      A     M      3.3;
      =     L     10.0;
      BLD   103;
      CALL FB    13 , DB    81 (
           EN_R                     := L     10.0,
           ID                       := W#16#1,
           R_ID                     := DW#16#1,
           NDR                      := DB2.DBX  100.0,
           ERROR                    := DB2.DBX  100.1,
           STATUS                   := DB2.DBW  102,
           RD_1                     := P#DB1.DBX0.0 BYTE 500,
           LEN                      := #RECV1_LEN);
      NOP   0;
NETWORK
TITLE =

      CALL SFC   20 (
           SRCBLK                   := P#M 5000.0 WORD 40,
           RET_VAL                  := #SFC20_RET_VAL,
           DSTBLK                   := P#DB21.DBX 0.0 WORD 40);
      NOP   0;
NETWORK
TITLE =

      L     80;
      T     #SEND1_LEN;
      NOP   0;
NETWORK
TITLE =LOCAL(CPU2) --> MAIN(CPU1) 공정상태

      A     M      0.2;
      =     L     10.0;
      BLD   103;
      AN    M      3.3;
      =     L     10.1;
      BLD   103;
      CALL FB    12 , DB    71 (
           REQ                      := L     10.0,
           R                        := L     10.1,
           ID                       := W#16#2,
           R_ID                     := DW#16#2,
           DONE                     := DB2.DBX    0.0,
           ERROR                    := DB2.DBX    0.1,
           STATUS                   := DB2.DBW    2,
           SD_1                     := P#DB21.DBX0.0 BYTE 80,
           LEN                      := #SEND1_LEN);
      NOP   0;
NETWORK
TITLE =

      L     80;
      T     #RECV2_LEN;
      NOP   0;
NETWORK
TITLE =MAIN(CPU1) --> LOCAL(CPU2) 셔틀상태
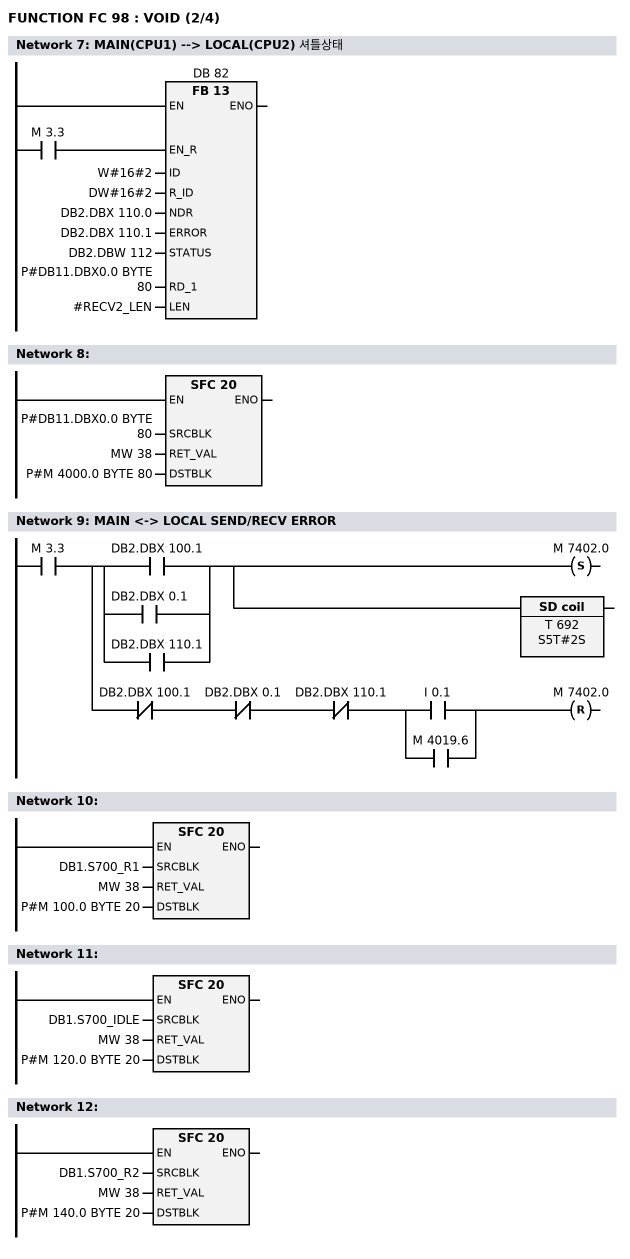

      A     M      3.3;
      =     L     10.0;
      BLD   103;
      CALL FB    13 , DB    82 (
           EN_R                     := L     10.0,
           ID                       := W#16#2,
           R_ID                     := DW#16#2,
           NDR                      := DB2.DBX  110.0,
           ERROR                    := DB2.DBX  110.1,
           STATUS                   := DB2.DBW  112,
           RD_1                     := P#DB11.DBX0.0 BYTE 80,
           LEN                      := #RECV2_LEN);
      NOP   0;
NETWORK
TITLE =

      CALL SFC   20 (
           SRCBLK                   := P#DB11.DBX0.0 BYTE 80,
           RET_VAL                  := MW    38,
           DSTBLK                   := P#M 4000.0 BYTE 80);
      NOP   0;
NETWORK
TITLE =MAIN <-> LOCAL SEND/RECV ERROR

      A     M      3.3;
      =     L     10.0;
      A     L     10.0;
      A(    ;
      O     DB2.DBX  100.1;
      O     DB2.DBX    0.1;
      O     DB2.DBX  110.1;
      )     ;
      S     M   7402.0;
      L     S5T#2S;
      SD    T    692;
      A     L     10.0;
      AN    DB2.DBX  100.1;
      AN    DB2.DBX    0.1;
      AN    DB2.DBX  110.1;
      A(    ;
      O     I      0.1;
      O     M   4019.6;
      )     ;
      R     M   7402.0;
NETWORK
TITLE =

      CALL SFC   20 (
           SRCBLK                   := DB1.S700_R1,
           RET_VAL                  := MW    38,
           DSTBLK                   := P#M 100.0 BYTE 20);
      NOP   0;
NETWORK
TITLE =

      CALL SFC   20 (
           SRCBLK                   := DB1.S700_IDLE,
           RET_VAL                  := MW    38,
           DSTBLK                   := P#M 120.0 BYTE 20);
      NOP   0;
NETWORK
TITLE =

      CALL SFC   20 (
           SRCBLK                   := DB1.S700_R2,
           RET_VAL                  := MW    38,
           DSTBLK                   := P#M 140.0 BYTE 20);
      NOP   0;
NETWORK
TITLE =
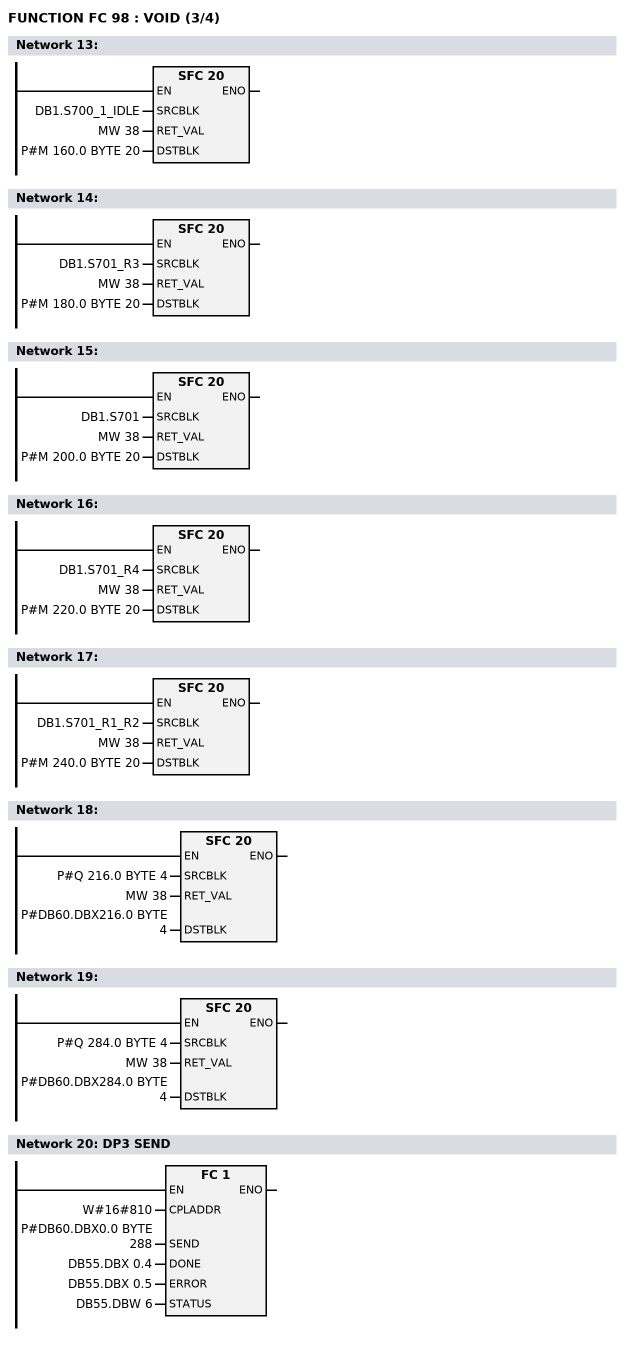

      CALL SFC   20 (
           SRCBLK                   := DB1.S700_1_IDLE,
           RET_VAL                  := MW    38,
           DSTBLK                   := P#M 160.0 BYTE 20);
      NOP   0;
NETWORK
TITLE =

      CALL SFC   20 (
           SRCBLK                   := DB1.S701_R3,
           RET_VAL                  := MW    38,
           DSTBLK                   := P#M 180.0 BYTE 20);
      NOP   0;
NETWORK
TITLE =

      CALL SFC   20 (
           SRCBLK                   := DB1.S701,
           RET_VAL                  := MW    38,
           DSTBLK                   := P#M 200.0 BYTE 20);
      NOP   0;
NETWORK
TITLE =

      CALL SFC   20 (
           SRCBLK                   := DB1.S701_R4,
           RET_VAL                  := MW    38,
           DSTBLK                   := P#M 220.0 BYTE 20);
      NOP   0;
NETWORK
TITLE =

      CALL SFC   20 (
           SRCBLK                   := DB1.S701_R1_R2,
           RET_VAL                  := MW    38,
           DSTBLK                   := P#M 240.0 BYTE 20);
      NOP   0;
NETWORK
TITLE =

      CALL SFC   20 (
           SRCBLK                   := P#Q 216.0 BYTE 4,
           RET_VAL                  := MW    38,
           DSTBLK                   := P#DB60.DBX216.0 BYTE 4);
      NOP   0;
NETWORK
TITLE =

      CALL SFC   20 (
           SRCBLK                   := P#Q 284.0 BYTE 4,
           RET_VAL                  := MW    38,
           DSTBLK                   := P#DB60.DBX284.0 BYTE 4);
      NOP   0;
NETWORK
TITLE =DP3 SEND

      CALL FC     1 (
           CPLADDR                  := W#16#810,
           SEND                     := P#DB60.DBX0.0 BYTE 288,
           DONE                     := DB55.DBX    0.4,
           ERROR                    := DB55.DBX    0.5,
           STATUS                   := DB55.DBW    6);
      NOP   0;
NETWORK
TITLE =DP3 RECV
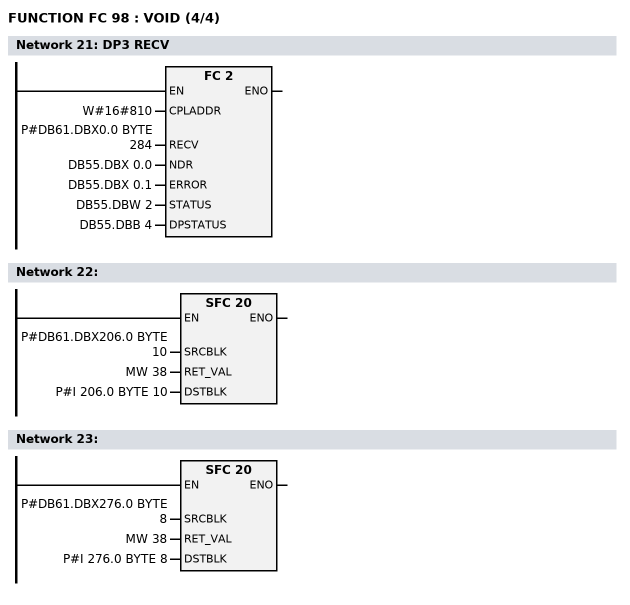

      CALL FC     2 (
           CPLADDR                  := W#16#810,
           RECV                     := P#DB61.DBX0.0 BYTE 284,
           NDR                      := DB55.DBX    0.0,
           ERROR                    := DB55.DBX    0.1,
           STATUS                   := DB55.DBW    2,
           DPSTATUS                 := DB55.DBB    4);
      NOP   0;
NETWORK
TITLE =

      CALL SFC   20 (
           SRCBLK                   := P#DB61.DBX206.0 BYTE 10,
           RET_VAL                  := MW    38,
           DSTBLK                   := P#I 206.0 BYTE 10);
      NOP   0;
NETWORK
TITLE =

      CALL SFC   20 (
           SRCBLK                   := P#DB61.DBX276.0 BYTE 8,
           RET_VAL                  := MW    38,
           DSTBLK                   := P#I 276.0 BYTE 8);
      NOP   0;
END_FUNCTION

FUNCTION FC 100 : VOID
TITLE =
VERSION : 0.1

BEGIN
NETWORK
TITLE =
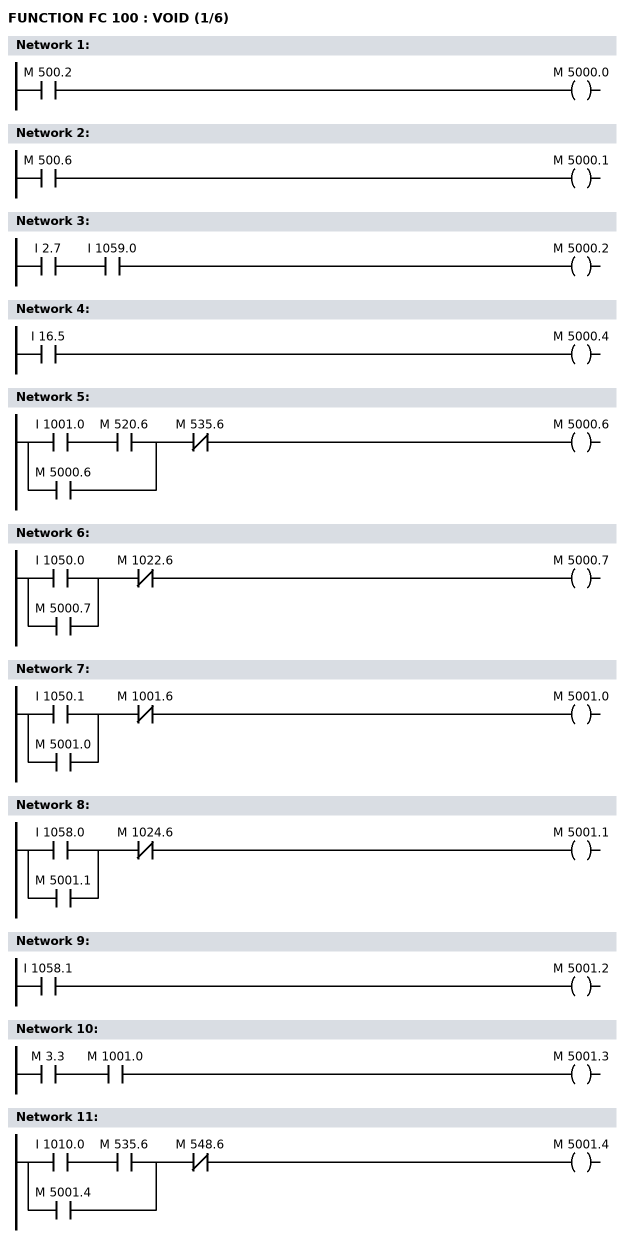

      A     M    500.2;
      =     M   5000.0;
NETWORK
TITLE =

      A     M    500.6;
      =     M   5000.1;
NETWORK
TITLE =

      A     I      2.7;
      A     I   1059.0;
      =     M   5000.2;
NETWORK
TITLE =

      A     I     16.5;
      =     M   5000.4;
NETWORK
TITLE =

      A(    ;
      A     I   1001.0;
      A     M    520.6;
      O     M   5000.6;
      )     ;
      AN    M    535.6;
      =     M   5000.6;
NETWORK
TITLE =

      A(    ;
      O     I   1050.0;
      O     M   5000.7;
      )     ;
      AN    M   1022.6;
      =     M   5000.7;
NETWORK
TITLE =

      A(    ;
      O     I   1050.1;
      O     M   5001.0;
      )     ;
      AN    M   1001.6;
      =     M   5001.0;
NETWORK
TITLE =

      A(    ;
      O     I   1058.0;
      O     M   5001.1;
      )     ;
      AN    M   1024.6;
      =     M   5001.1;
NETWORK
TITLE =

      A     I   1058.1;
      =     M   5001.2;
NETWORK
TITLE =

      A     M      3.3;
      A     M   1001.0;
      =     M   5001.3;
NETWORK
TITLE =

      A(    ;
      A     I   1010.0;
      A     M    535.6;
      O     M   5001.4;
      )     ;
      AN    M    548.6;
      =     M   5001.4;
NETWORK
TITLE =
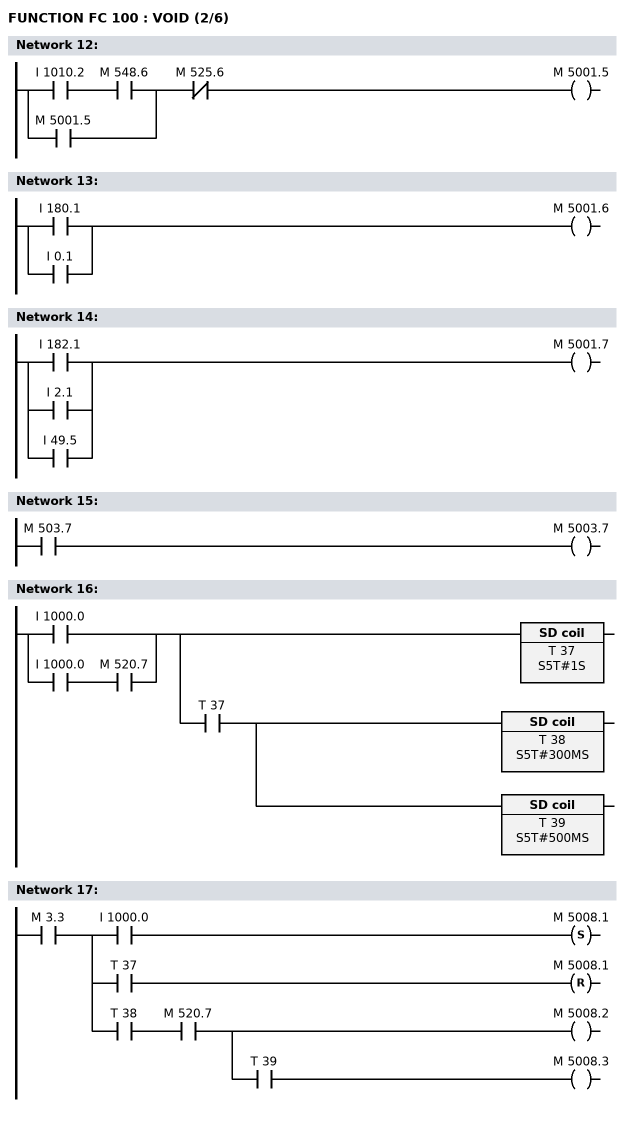

      A(    ;
      A     I   1010.2;
      A     M    548.6;
      O     M   5001.5;
      )     ;
      AN    M    525.6;
      =     M   5001.5;
NETWORK
TITLE =

      O     I    180.1;
      O     I      0.1;
      =     M   5001.6;
NETWORK
TITLE =

      O     I    182.1;
      O     I      2.1;
      O     I     49.5;
      =     M   5001.7;
NETWORK
TITLE =

      A     M    503.7;
      =     M   5003.7;
NETWORK
TITLE =

      O     I   1000.0;
      O     ;
      A     I   1000.0;
      A     M    520.7;
      =     L      0.0;
      A     L      0.0;
      BLD   102;
      L     S5T#1S;
      SD    T     37;
      A     L      0.0;
      A     T     37;
      L     S5T#300MS;
      SD    T     38;
      L     S5T#500MS;
      SD    T     39;
NETWORK
TITLE =

      A     M      3.3;
      =     L      0.0;
      A     L      0.0;
      A     I   1000.0;
      S     M   5008.1;
      A     L      0.0;
      A     T     37;
      R     M   5008.1;
      A     L      0.0;
      A     T     38;
      A     M    520.7;
      =     L      0.1;
      A     L      0.1;
      BLD   102;
      =     M   5008.2;
      A     L      0.1;
      A     T     39;
      =     M   5008.3;
NETWORK
TITLE =
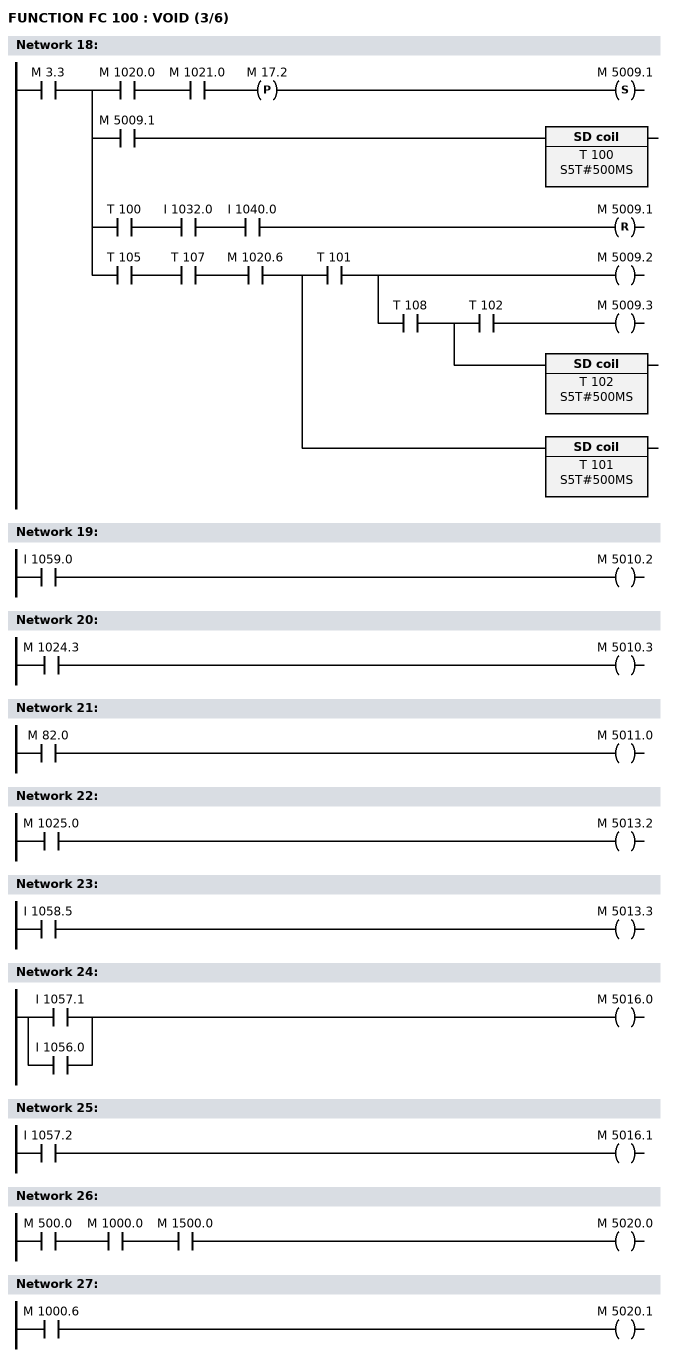

      A     M      3.3;
      =     L      0.0;
      A     L      0.0;
      A     M   1020.0;
      A     M   1021.0;
      FP    M     17.2;
      S     M   5009.1;
      A     L      0.0;
      A     M   5009.1;
      L     S5T#500MS;
      SD    T    100;
      A     L      0.0;
      A     T    100;
      A     I   1032.0;
      A     I   1040.0;
      R     M   5009.1;
      A     L      0.0;
      A     T    105;
      A     T    107;
      A     M   1020.6;
      =     L      0.1;
      A     L      0.1;
      A     T    101;
      =     L      0.2;
      A     L      0.2;
      BLD   102;
      =     M   5009.2;
      A     L      0.2;
      A     T    108;
      =     L      0.3;
      A     L      0.3;
      A     T    102;
      =     M   5009.3;
      A     L      0.3;
      BLD   102;
      L     S5T#500MS;
      SD    T    102;
      A     L      0.1;
      BLD   102;
      L     S5T#500MS;
      SD    T    101;
NETWORK
TITLE =

      A     I   1059.0;
      =     M   5010.2;
NETWORK
TITLE =

      A     M   1024.3;
      =     M   5010.3;
NETWORK
TITLE =

      A     M     82.0;
      =     M   5011.0;
NETWORK
TITLE =

      A     M   1025.0;
      =     M   5013.2;
NETWORK
TITLE =

      A     I   1058.5;
      =     M   5013.3;
NETWORK
TITLE =

      O     I   1057.1;
      O     I   1056.0;
      =     M   5016.0;
NETWORK
TITLE =

      A     I   1057.2;
      =     M   5016.1;
NETWORK
TITLE =

      A     M    500.0;
      A     M   1000.0;
      A     M   1500.0;
      =     M   5020.0;
NETWORK
TITLE =

      A     M   1000.6;
      =     M   5020.1;
NETWORK
TITLE =
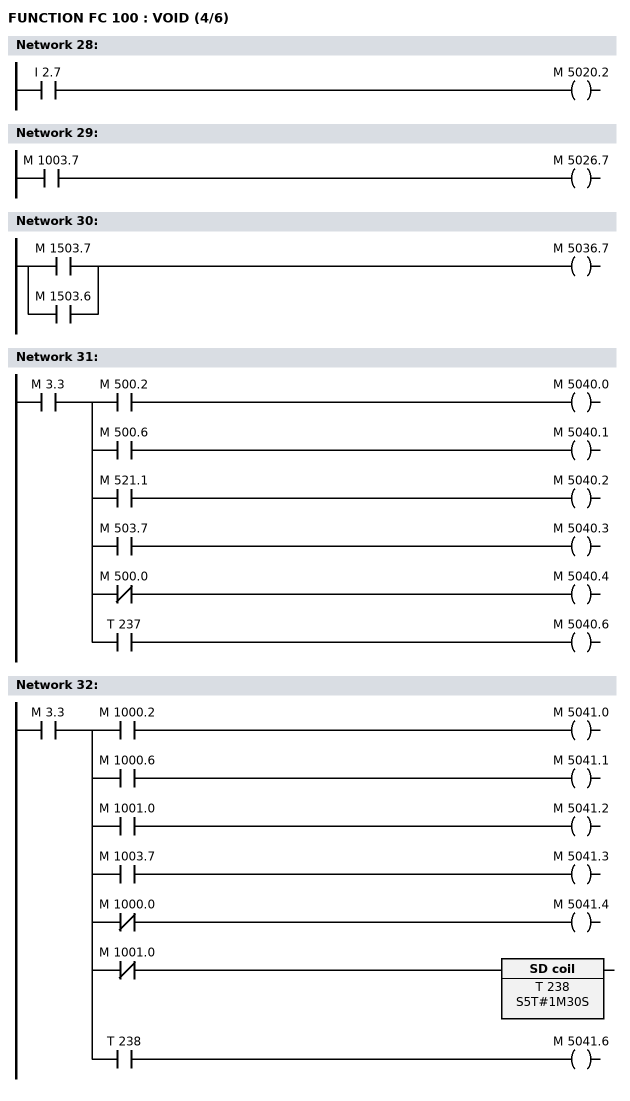

      A     I      2.7;
      =     M   5020.2;
NETWORK
TITLE =

      A     M   1003.7;
      =     M   5026.7;
NETWORK
TITLE =

      O     M   1503.7;
      O     M   1503.6;
      =     M   5036.7;
NETWORK
TITLE =

      A     M      3.3;
      =     L      0.0;
      A     L      0.0;
      A     M    500.2;
      =     M   5040.0;
      A     L      0.0;
      A     M    500.6;
      =     M   5040.1;
      A     L      0.0;
      A     M    521.1;
      =     M   5040.2;
      A     L      0.0;
      A     M    503.7;
      =     M   5040.3;
      A     L      0.0;
      AN    M    500.0;
      =     M   5040.4;
      A     L      0.0;
      A     T    237;
      =     M   5040.6;
NETWORK
TITLE =

      A     M      3.3;
      =     L      0.0;
      A     L      0.0;
      A     M   1000.2;
      =     M   5041.0;
      A     L      0.0;
      A     M   1000.6;
      =     M   5041.1;
      A     L      0.0;
      A     M   1001.0;
      =     M   5041.2;
      A     L      0.0;
      A     M   1003.7;
      =     M   5041.3;
      A     L      0.0;
      AN    M   1000.0;
      =     M   5041.4;
      A     L      0.0;
      AN    M   1001.0;
      L     S5T#1M30S;
      SD    T    238;
      A     L      0.0;
      A     T    238;
      =     M   5041.6;
NETWORK
TITLE =
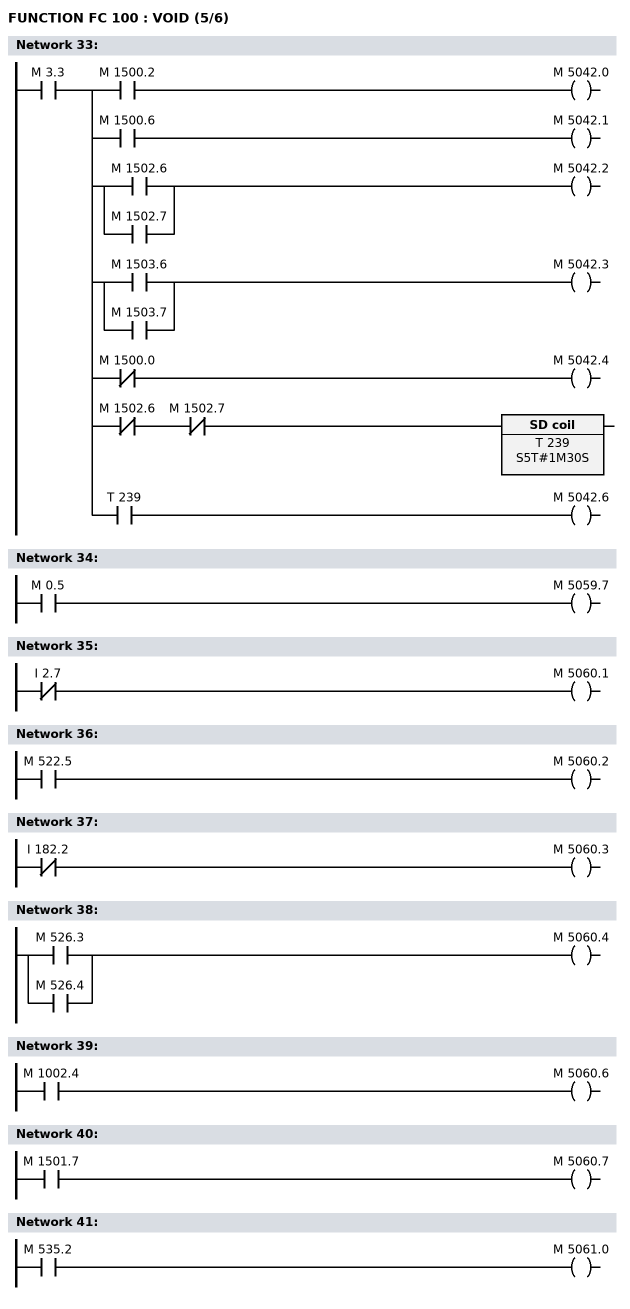

      A     M      3.3;
      =     L      0.0;
      A     L      0.0;
      A     M   1500.2;
      =     M   5042.0;
      A     L      0.0;
      A     M   1500.6;
      =     M   5042.1;
      A     L      0.0;
      A(    ;
      O     M   1502.6;
      O     M   1502.7;
      )     ;
      =     M   5042.2;
      A     L      0.0;
      A(    ;
      O     M   1503.6;
      O     M   1503.7;
      )     ;
      =     M   5042.3;
      A     L      0.0;
      AN    M   1500.0;
      =     M   5042.4;
      A     L      0.0;
      AN    M   1502.6;
      AN    M   1502.7;
      L     S5T#1M30S;
      SD    T    239;
      A     L      0.0;
      A     T    239;
      =     M   5042.6;
NETWORK
TITLE =

      A     M      0.5;
      =     M   5059.7;
NETWORK
TITLE =

      AN    I      2.7;
      =     M   5060.1;
NETWORK
TITLE =

      A     M    522.5;
      =     M   5060.2;
NETWORK
TITLE =

      AN    I    182.2;
      =     M   5060.3;
NETWORK
TITLE =

      O     M    526.3;
      O     M    526.4;
      =     M   5060.4;
NETWORK
TITLE =

      A     M   1002.4;
      =     M   5060.6;
NETWORK
TITLE =

      A     M   1501.7;
      =     M   5060.7;
NETWORK
TITLE =

      A     M    535.2;
      =     M   5061.0;
NETWORK
TITLE =
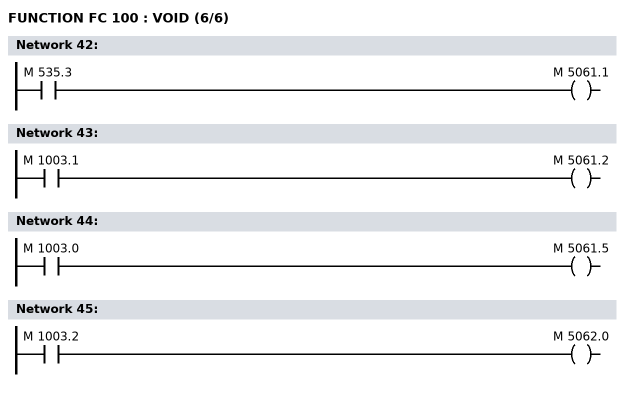

      A     M    535.3;
      =     M   5061.1;
NETWORK
TITLE =

      A     M   1003.1;
      =     M   5061.2;
NETWORK
TITLE =

      A     M   1003.0;
      =     M   5061.5;
NETWORK
TITLE =

      A     M   1003.2;
      =     M   5062.0;
NETWORK
TITLE =

      AN    OV;
      A(    ;
      O     T    158;
      O     T    159;
      O     T    160;
      O     T    161;
      O     T    164;
      O     T    165;
      O     T    166;
      O     T    167;
      )     ;
      =     M   5063.7;
NETWORK
TITLE =
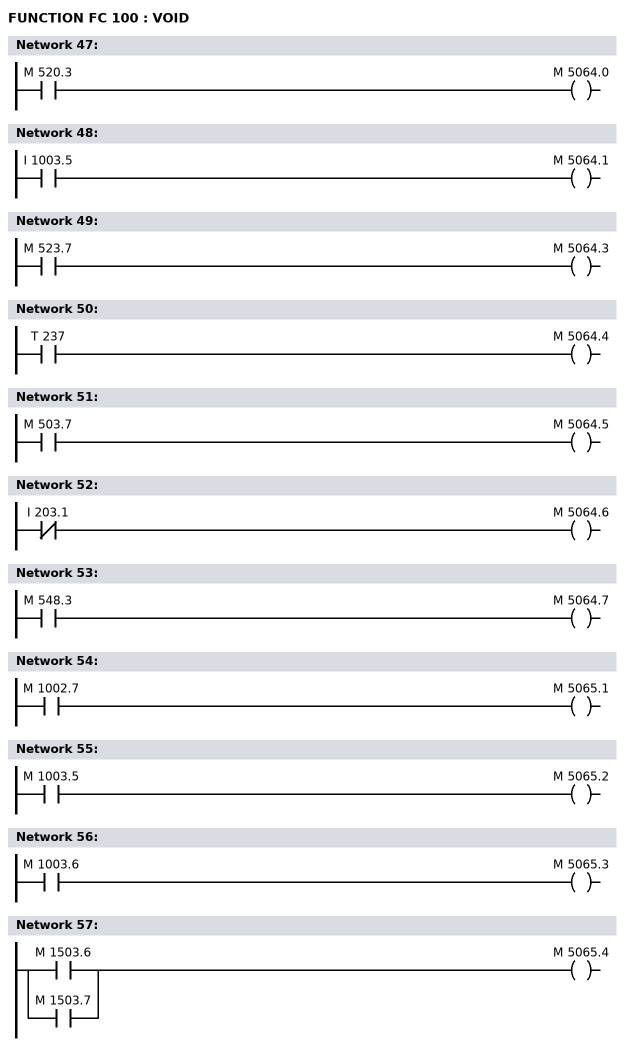

      A     M    520.3;
      =     M   5064.0;
NETWORK
TITLE =

      A     I   1003.5;
      =     M   5064.1;
NETWORK
TITLE =

      A     M    523.7;
      =     M   5064.3;
NETWORK
TITLE =

      A     T    237;
      =     M   5064.4;
NETWORK
TITLE =

      A     M    503.7;
      =     M   5064.5;
NETWORK
TITLE =

      AN    I    203.1;
      =     M   5064.6;
NETWORK
TITLE =

      A     M    548.3;
      =     M   5064.7;
NETWORK
TITLE =

      A     M   1002.7;
      =     M   5065.1;
NETWORK
TITLE =

      A     M   1003.5;
      =     M   5065.2;
NETWORK
TITLE =

      A     M   1003.6;
      =     M   5065.3;
NETWORK
TITLE =

      O     M   1503.6;
      O     M   1503.7;
      =     M   5065.4;
NETWORK
TITLE =

      AN    OV;
      =     L      0.0;
      A     L      0.0;
      A     M    522.3;
      =     M   5066.0;
      A     L      0.0;
      A     M    523.3;
      =     M   5066.1;
      A     L      0.0;
      A(    ;
      O     M   1020.3;
      O     M   1022.3;
      )     ;
      =     M   5066.2;
      A     L      0.0;
      A(    ;
      O     M   1021.3;
      O     M   1024.3;
      )     ;
      =     M   5066.3;
NETWORK
TITLE =

      AN    OV;
      =     L      0.0;
      A     L      0.0;
      A     M    521.2;
      =     M   5066.4;
      A     L      0.0;
      A     I   1010.4;
      =     M   5066.6;
      A     L      0.0;
      AN    T    232;
      AN    T    233;
      NOT   ;
      =     M   5066.7;
NETWORK
TITLE =

      AN    OV;
      =     L      0.0;
      A     L      0.0;
      A     I      2.1;
      =     M   5067.1;
      A     L      0.0;
      A     I    182.1;
      =     M   5067.2;
      A     L      0.0;
      A     M   1002.5;
      =     M   5067.3;
      A     L      0.0;
      A     I    279.0;
      A     M   1052.7;
      A     M   1053.1;
      =     M   5067.4;
      A     L      0.0;
      A     I     49.5;
      =     M   5067.5;
      A     L      0.0;
      A(    ;
      ON    I     16.5;
      ON    I     16.0;
      )     ;
      =     M   5067.6;
NETWORK
TITLE =

      AN    OV;
      =     L      0.0;
      A     L      0.0;
      A     M   1003.3;
      =     M   5068.1;
      A     L      0.0;
      A     M   1018.7;
      =     M   5068.2;
NETWORK
TITLE =

      A     I   1034.5;
      =     M   5068.7;
NETWORK
TITLE =

      AN    OV;
      =     L      0.0;
      A     L      0.0;
      A(    ;
      O     M   1100.0;
      O     M   1100.1;
      )     ;
      =     M   5069.0;
      A     L      0.0;
      A(    ;
      O     M   1100.4;
      O     M   1100.5;
      )     ;
      =     M   5069.1;
NETWORK
TITLE =
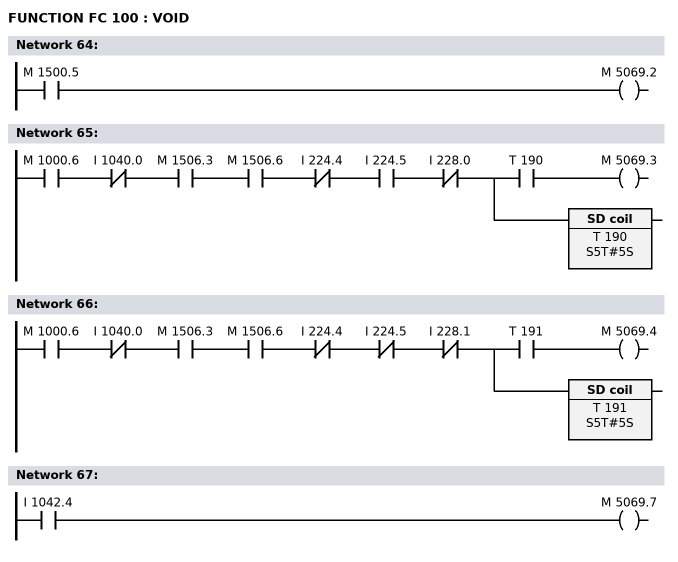

      A     M   1500.5;
      =     M   5069.2;
NETWORK
TITLE =

      A     M   1000.6;
      AN    I   1040.0;
      A     M   1506.3;
      A     M   1506.6;
      AN    I    224.4;
      A     I    224.5;
      AN    I    228.0;
      =     L      0.0;
      A     L      0.0;
      A     T    190;
      =     M   5069.3;
      A     L      0.0;
      BLD   102;
      L     S5T#5S;
      SD    T    190;
NETWORK
TITLE =

      A     M   1000.6;
      AN    I   1040.0;
      A     M   1506.3;
      A     M   1506.6;
      AN    I    224.4;
      AN    I    224.5;
      AN    I    228.1;
      =     L      0.0;
      A     L      0.0;
      A     T    191;
      =     M   5069.4;
      A     L      0.0;
      BLD   102;
      L     S5T#5S;
      SD    T    191;
NETWORK
TITLE =

      A     I   1042.4;
      =     M   5069.7;
END_FUNCTION

FUNCTION_BLOCK FB 105
TITLE =
VERSION : 0.1


VAR
  MW_0_BUFF : ARRAY  [0 .. 59 ] OF WORD ;
  S701_RBT1_WELD_OK_PLS : BOOL ;
  S701_RBT1_WELD_NG_PLS : BOOL ;
  S701_RBT1_WELD_PASS_PLS : BOOL ;
  S701_RBT2_WELD_OK_PLS : BOOL ;
  S701_RBT2_WELD_NG_PLS : BOOL ;
  S701_RBT2_WELD_PASS_PLS : BOOL ;
  S701_CHECK_SUM_PLS : BOOL ;
  S701_WELD_DATA_MOV_BUFF : BOOL ;
  PLS1 : BOOL ;
  PLS2 : BOOL ;
END_VAR
VAR_TEMP
  SFC20_RET_VAL : INT ;
END_VAR
BEGIN
NETWORK
TITLE =MES 용접누락 DATA -> #701차종코드(2011) 기준값 버퍼로 전송(LM)
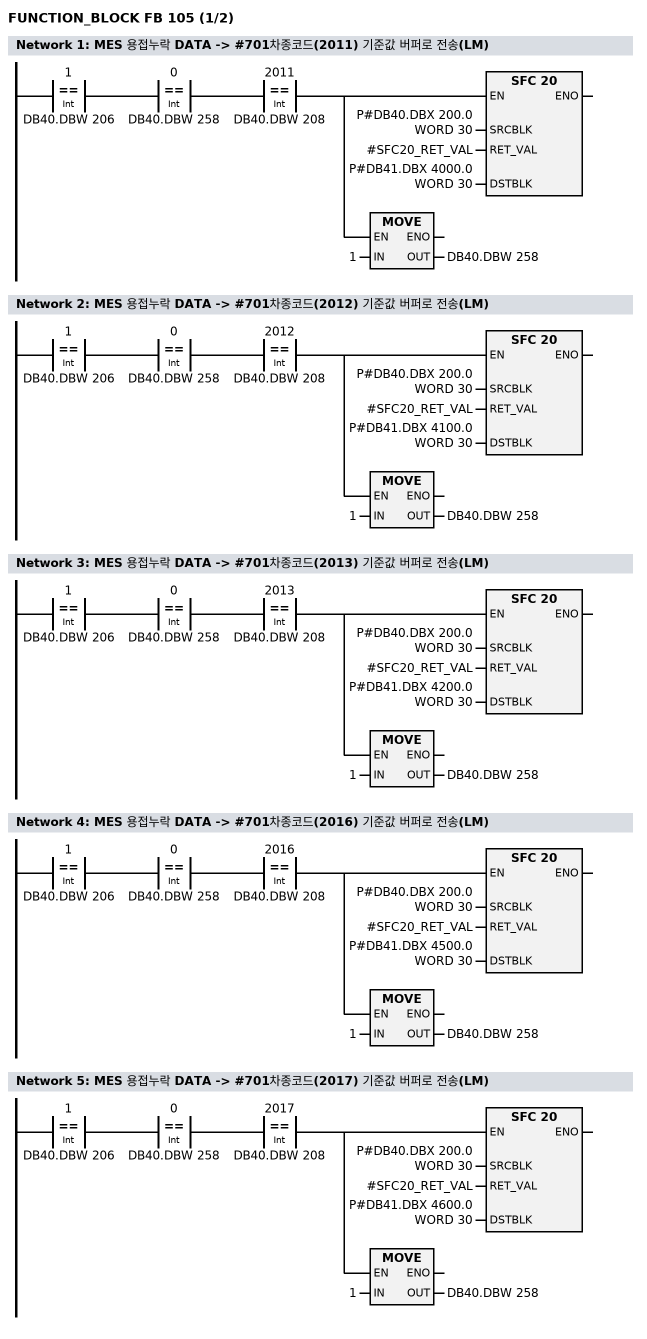

      A(    ;
      L     1;
      L     DB40.DBW  206;
      ==I   ;
      )     ;
      A(    ;
      L     0;
      L     DB40.DBW  258;
      ==I   ;
      )     ;
      A(    ;
      L     2011;
      L     DB40.DBW  208;
      ==I   ;
      )     ;
      =     L      2.0;
      A     L      2.0;
      JNB   _001;
      CALL SFC   20 (
           SRCBLK                   := P#DB40.DBX 200.0 WORD 30,
           RET_VAL                  := #SFC20_RET_VAL,
           DSTBLK                   := P#DB41.DBX 4000.0 WORD 30);
_001: NOP   0;
      A     L      2.0;
      JNB   _002;
      L     1;
      T     DB40.DBW  258;
_002: NOP   0;
NETWORK
TITLE =MES 용접누락 DATA -> #701차종코드(2012) 기준값 버퍼로 전송(LM)

      A(    ;
      L     1;
      L     DB40.DBW  206;
      ==I   ;
      )     ;
      A(    ;
      L     0;
      L     DB40.DBW  258;
      ==I   ;
      )     ;
      A(    ;
      L     2012;
      L     DB40.DBW  208;
      ==I   ;
      )     ;
      =     L      2.0;
      A     L      2.0;
      JNB   _003;
      CALL SFC   20 (
           SRCBLK                   := P#DB40.DBX 200.0 WORD 30,
           RET_VAL                  := #SFC20_RET_VAL,
           DSTBLK                   := P#DB41.DBX 4100.0 WORD 30);
_003: NOP   0;
      A     L      2.0;
      JNB   _004;
      L     1;
      T     DB40.DBW  258;
_004: NOP   0;
NETWORK
TITLE =MES 용접누락 DATA -> #701차종코드(2013) 기준값 버퍼로 전송(LM)
//
//
      A(    ;
      L     1;
      L     DB40.DBW  206;
      ==I   ;
      )     ;
      A(    ;
      L     0;
      L     DB40.DBW  258;
      ==I   ;
      )     ;
      A(    ;
      L     2013;
      L     DB40.DBW  208;
      ==I   ;
      )     ;
      =     L      2.0;
      A     L      2.0;
      JNB   _005;
      CALL SFC   20 (
           SRCBLK                   := P#DB40.DBX 200.0 WORD 30,
           RET_VAL                  := #SFC20_RET_VAL,
           DSTBLK                   := P#DB41.DBX 4200.0 WORD 30);
_005: NOP   0;
      A     L      2.0;
      JNB   _006;
      L     1;
      T     DB40.DBW  258;
_006: NOP   0;
NETWORK
TITLE =MES 용접누락 DATA -> #701차종코드(2016) 기준값 버퍼로 전송(LM)

      A(    ;
      L     1;
      L     DB40.DBW  206;
      ==I   ;
      )     ;
      A(    ;
      L     0;
      L     DB40.DBW  258;
      ==I   ;
      )     ;
      A(    ;
      L     2016;
      L     DB40.DBW  208;
      ==I   ;
      )     ;
      =     L      2.0;
      A     L      2.0;
      JNB   _007;
      CALL SFC   20 (
           SRCBLK                   := P#DB40.DBX 200.0 WORD 30,
           RET_VAL                  := #SFC20_RET_VAL,
           DSTBLK                   := P#DB41.DBX 4500.0 WORD 30);
_007: NOP   0;
      A     L      2.0;
      JNB   _008;
      L     1;
      T     DB40.DBW  258;
_008: NOP   0;
NETWORK
TITLE =MES 용접누락 DATA -> #701차종코드(2017) 기준값 버퍼로 전송(LM)

      A(    ;
      L     1;
      L     DB40.DBW  206;
      ==I   ;
      )     ;
      A(    ;
      L     0;
      L     DB40.DBW  258;
      ==I   ;
      )     ;
      A(    ;
      L     2017;
      L     DB40.DBW  208;
      ==I   ;
      )     ;
      =     L      2.0;
      A     L      2.0;
      JNB   _009;
      CALL SFC   20 (
           SRCBLK                   := P#DB40.DBX 200.0 WORD 30,
           RET_VAL                  := #SFC20_RET_VAL,
           DSTBLK                   := P#DB41.DBX 4600.0 WORD 30);
_009: NOP   0;
      A     L      2.0;
      JNB   _00a;
      L     1;
      T     DB40.DBW  258;
_00a: NOP   0;
NETWORK
TITLE =MES 용접누락 DATA -> #701차종코드(2018) 기준값 버퍼로 전송(LM)
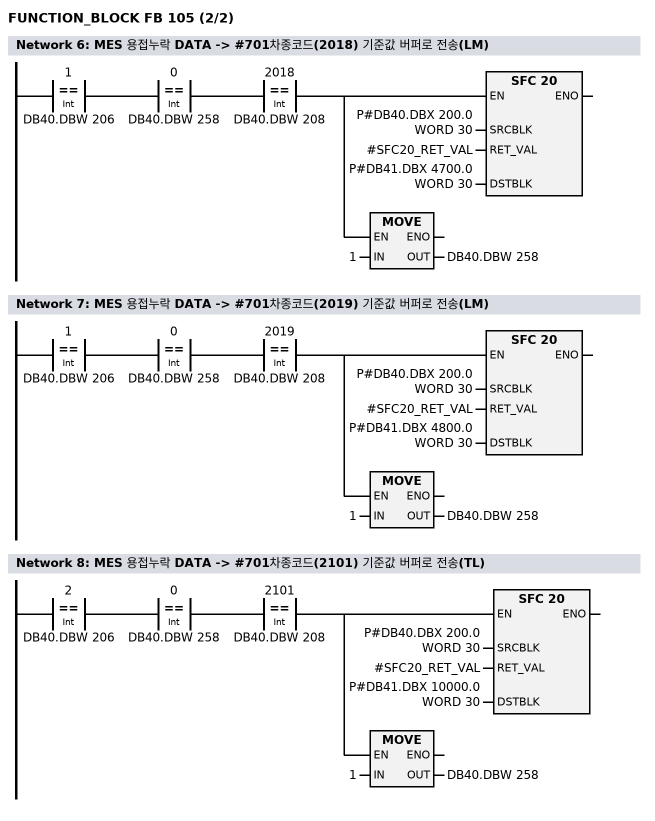

      A(    ;
      L     1;
      L     DB40.DBW  206;
      ==I   ;
      )     ;
      A(    ;
      L     0;
      L     DB40.DBW  258;
      ==I   ;
      )     ;
      A(    ;
      L     2018;
      L     DB40.DBW  208;
      ==I   ;
      )     ;
      =     L      2.0;
      A     L      2.0;
      JNB   _00b;
      CALL SFC   20 (
           SRCBLK                   := P#DB40.DBX 200.0 WORD 30,
           RET_VAL                  := #SFC20_RET_VAL,
           DSTBLK                   := P#DB41.DBX 4700.0 WORD 30);
_00b: NOP   0;
      A     L      2.0;
      JNB   _00c;
      L     1;
      T     DB40.DBW  258;
_00c: NOP   0;
NETWORK
TITLE =MES 용접누락 DATA -> #701차종코드(2019) 기준값 버퍼로 전송(LM)

      A(    ;
      L     1;
      L     DB40.DBW  206;
      ==I   ;
      )     ;
      A(    ;
      L     0;
      L     DB40.DBW  258;
      ==I   ;
      )     ;
      A(    ;
      L     2019;
      L     DB40.DBW  208;
      ==I   ;
      )     ;
      =     L      2.0;
      A     L      2.0;
      JNB   _00d;
      CALL SFC   20 (
           SRCBLK                   := P#DB40.DBX 200.0 WORD 30,
           RET_VAL                  := #SFC20_RET_VAL,
           DSTBLK                   := P#DB41.DBX 4800.0 WORD 30);
_00d: NOP   0;
      A     L      2.0;
      JNB   _00e;
      L     1;
      T     DB40.DBW  258;
_00e: NOP   0;
NETWORK
TITLE =MES 용접누락 DATA -> #701차종코드(2101) 기준값 버퍼로 전송(TL)

      A(    ;
      L     2;
      L     DB40.DBW  206;
      ==I   ;
      )     ;
      A(    ;
      L     0;
      L     DB40.DBW  258;
      ==I   ;
      )     ;
      A(    ;
      L     2101;
      L     DB40.DBW  208;
      ==I   ;
      )     ;
      =     L      2.0;
      A     L      2.0;
      JNB   _00f;
      CALL SFC   20 (
           SRCBLK                   := P#DB40.DBX 200.0 WORD 30,
           RET_VAL                  := #SFC20_RET_VAL,
           DSTBLK                   := P#DB41.DBX 10000.0 WORD 30);
_00f: NOP   0;
      A     L      2.0;
      JNB   _010;
      L     1;
      T     DB40.DBW  258;
_010: NOP   0;
NETWORK
TITLE =#701 RBT1호 용접카운터 INT -> DB로 전송보조

      AN    OV;
      =     L      2.0;
      A     L      2.0;
      A     I   1036.0;
      =     M     11.0;
      A     L      2.0;
      A     I   1036.1;
      =     M     11.1;
      A     L      2.0;
      A     I   1036.2;
      =     M     11.2;
      A     L      2.0;
      A     I   1036.3;
      =     M     11.3;
      A     L      2.0;
      A     I   1036.4;
      =     M     11.4;
      A     L      2.0;
      A     OV;
      =     M     11.5;
      =     M     11.6;
      =     M     11.7;
NETWORK
TITLE =#701 RBT1호 용접카운터 INT -> DB로 전송
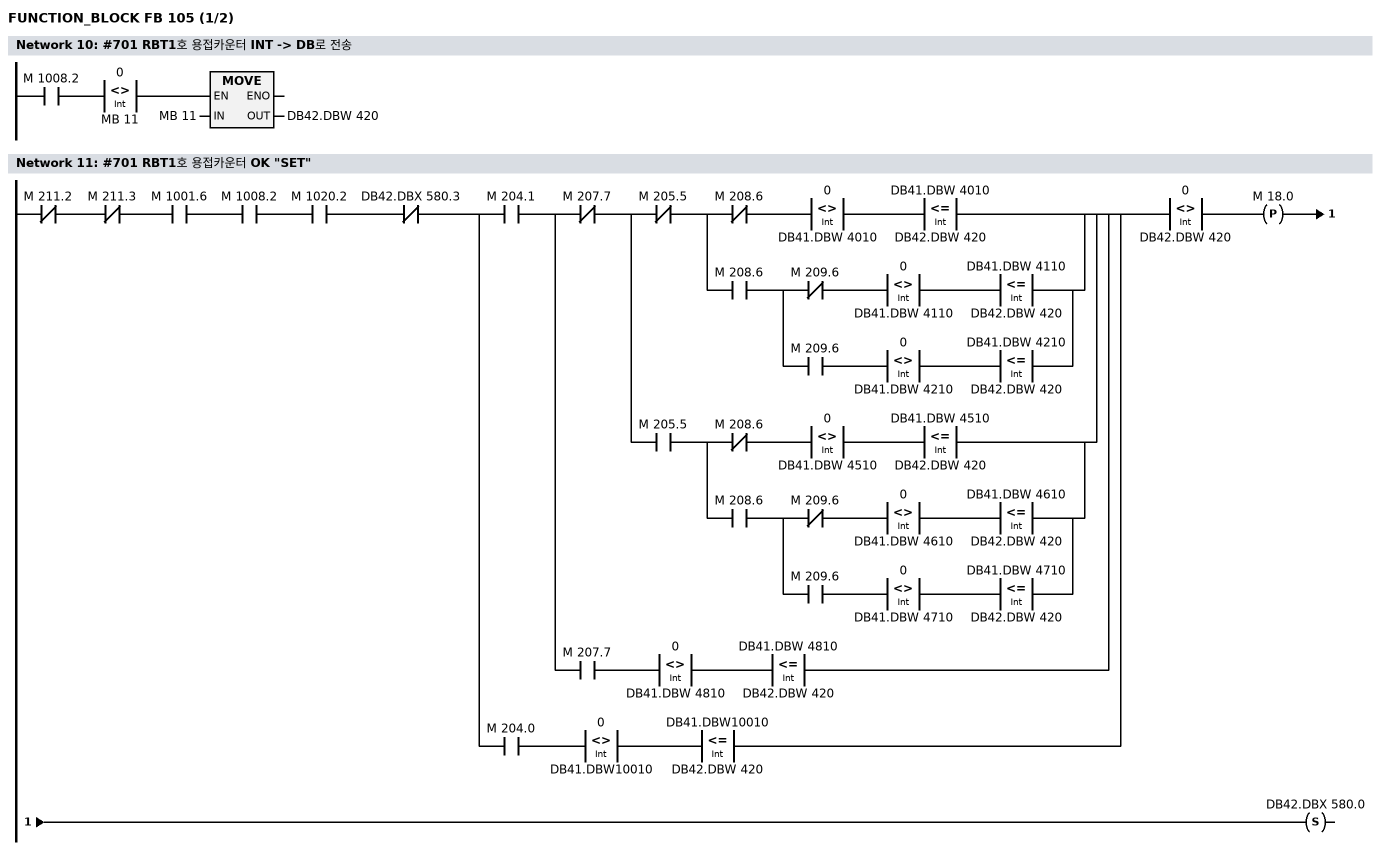

      A     M   1008.2;
      A(    ;
      L     0;
      L     MB    11;
      <>I   ;
      )     ;
      JNB   _011;
      L     MB    11;
      T     DB42.DBW  420;
_011: NOP   0;
NETWORK
TITLE =#701 RBT1호 용접카운터 OK "SET"

      AN    M    211.2;
      AN    M    211.3;
      A     M   1001.6;
      A     M   1008.2;
      A     M   1020.2;
      AN    DB42.DBX  580.3;
      A(    ;
      A     M    204.1;
      A(    ;
      AN    M    207.7;
      A(    ;
      AN    M    205.5;
      A(    ;
      AN    M    208.6;
      A(    ;
      L     0;
      L     DB41.DBW 4010;
      <>I   ;
      )     ;
      A(    ;
      L     DB41.DBW 4010;
      L     DB42.DBW  420;
      <=I   ;
      )     ;
      O     ;
      A     M    208.6;
      A(    ;
      AN    M    209.6;
      A(    ;
      L     0;
      L     DB41.DBW 4110;
      <>I   ;
      )     ;
      A(    ;
      L     DB41.DBW 4110;
      L     DB42.DBW  420;
      <=I   ;
      )     ;
      O     ;
      A     M    209.6;
      A(    ;
      L     0;
      L     DB41.DBW 4210;
      <>I   ;
      )     ;
      A(    ;
      L     DB41.DBW 4210;
      L     DB42.DBW  420;
      <=I   ;
      )     ;
      )     ;
      )     ;
      O     ;
      A     M    205.5;
      A(    ;
      AN    M    208.6;
      A(    ;
      L     0;
      L     DB41.DBW 4510;
      <>I   ;
      )     ;
      A(    ;
      L     DB41.DBW 4510;
      L     DB42.DBW  420;
      <=I   ;
      )     ;
      O     ;
      A     M    208.6;
      A(    ;
      AN    M    209.6;
      A(    ;
      L     0;
      L     DB41.DBW 4610;
      <>I   ;
      )     ;
      A(    ;
      L     DB41.DBW 4610;
      L     DB42.DBW  420;
      <=I   ;
      )     ;
      O     ;
      A     M    209.6;
      A(    ;
      L     0;
      L     DB41.DBW 4710;
      <>I   ;
      )     ;
      A(    ;
      L     DB41.DBW 4710;
      L     DB42.DBW  420;
      <=I   ;
      )     ;
      )     ;
      )     ;
      )     ;
      O     ;
      A     M    207.7;
      A(    ;
      L     0;
      L     DB41.DBW 4810;
      <>I   ;
      )     ;
      A(    ;
      L     DB41.DBW 4810;
      L     DB42.DBW  420;
      <=I   ;
      )     ;
      )     ;
      O     ;
      A     M    204.0;
      A(    ;
      L     0;
      L     DB41.DBW10010;
      <>I   ;
      )     ;
      A(    ;
      L     DB41.DBW10010;
      L     DB42.DBW  420;
      <=I   ;
      )     ;
      )     ;
      A(    ;
      L     0;
      L     DB42.DBW  420;
      <>I   ;
      )     ;
      FP    M     18.0;
      S     DB42.DBX  580.0;
NETWORK
TITLE =#701 RBT1호 용접카운터 NG "SET"
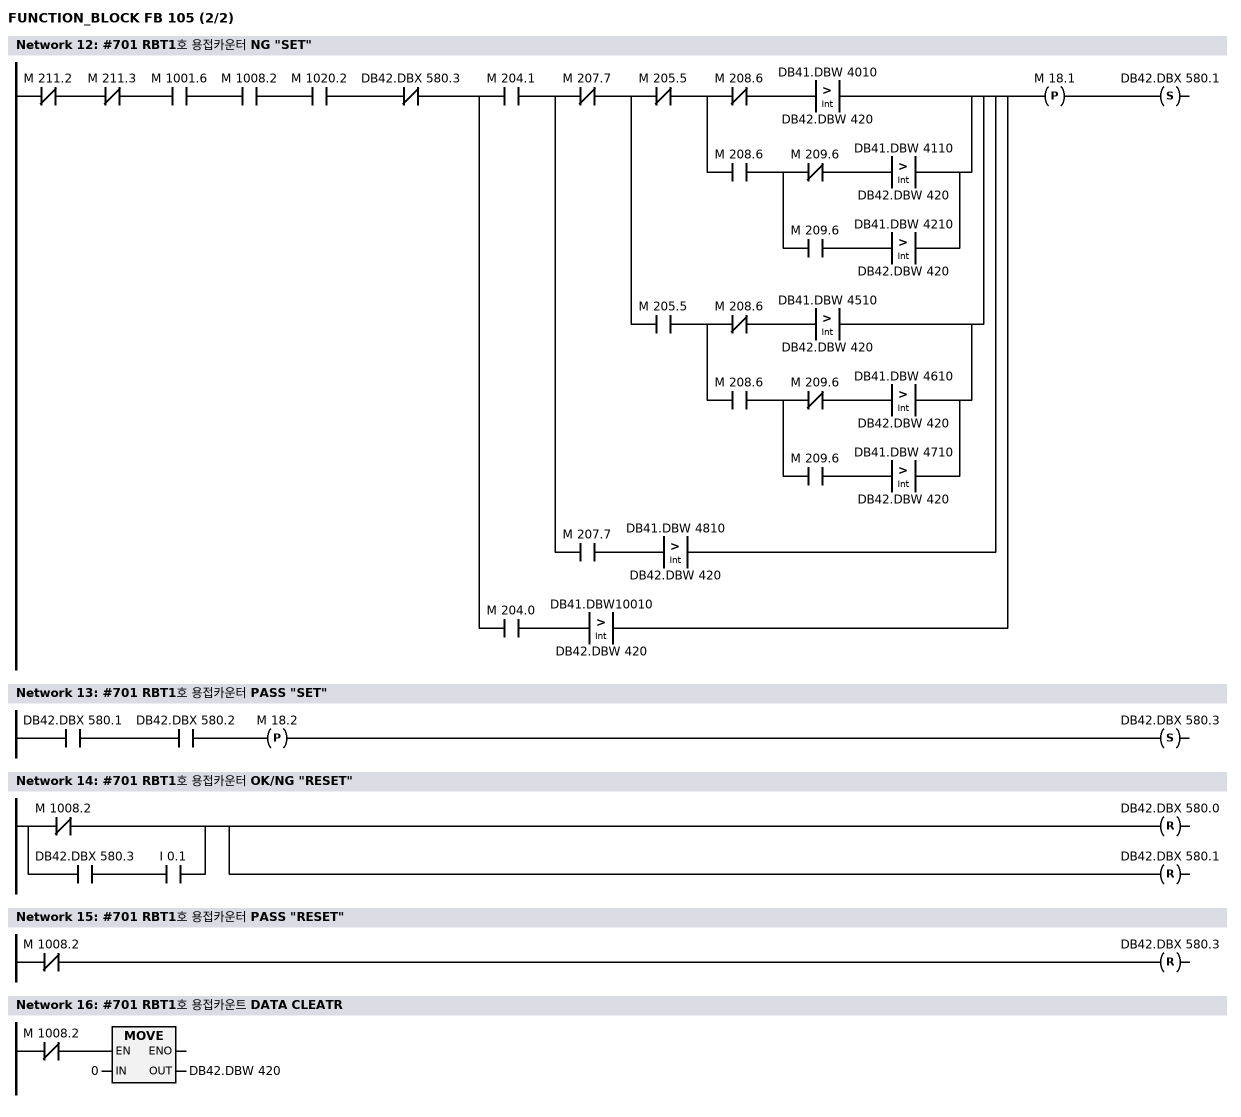

      AN    M    211.2;
      AN    M    211.3;
      A     M   1001.6;
      A     M   1008.2;
      A     M   1020.2;
      AN    DB42.DBX  580.3;
      A(    ;
      A     M    204.1;
      A(    ;
      AN    M    207.7;
      A(    ;
      AN    M    205.5;
      A(    ;
      AN    M    208.6;
      A(    ;
      L     DB41.DBW 4010;
      L     DB42.DBW  420;
      >I    ;
      )     ;
      O     ;
      A     M    208.6;
      A(    ;
      AN    M    209.6;
      A(    ;
      L     DB41.DBW 4110;
      L     DB42.DBW  420;
      >I    ;
      )     ;
      O     ;
      A     M    209.6;
      A(    ;
      L     DB41.DBW 4210;
      L     DB42.DBW  420;
      >I    ;
      )     ;
      )     ;
      )     ;
      O     ;
      A     M    205.5;
      A(    ;
      AN    M    208.6;
      A(    ;
      L     DB41.DBW 4510;
      L     DB42.DBW  420;
      >I    ;
      )     ;
      O     ;
      A     M    208.6;
      A(    ;
      AN    M    209.6;
      A(    ;
      L     DB41.DBW 4610;
      L     DB42.DBW  420;
      >I    ;
      )     ;
      O     ;
      A     M    209.6;
      A(    ;
      L     DB41.DBW 4710;
      L     DB42.DBW  420;
      >I    ;
      )     ;
      )     ;
      )     ;
      )     ;
      O     ;
      A     M    207.7;
      A(    ;
      L     DB41.DBW 4810;
      L     DB42.DBW  420;
      >I    ;
      )     ;
      )     ;
      O     ;
      A     M    204.0;
      A(    ;
      L     DB41.DBW10010;
      L     DB42.DBW  420;
      >I    ;
      )     ;
      )     ;
      FP    M     18.1;
      S     DB42.DBX  580.1;
NETWORK
TITLE =#701 RBT1호 용접카운터 PASS "SET"

      A     DB42.DBX  580.1;
      A     DB42.DBX  580.2;
      FP    M     18.2;
      S     DB42.DBX  580.3;
NETWORK
TITLE =#701 RBT1호 용접카운터 OK/NG "RESET"

      ON    M   1008.2;
      O     ;
      A     DB42.DBX  580.3;
      A     I      0.1;
      R     DB42.DBX  580.0;
      R     DB42.DBX  580.1;
NETWORK
TITLE =#701 RBT1호 용접카운터 PASS "RESET"

      AN    M   1008.2;
      R     DB42.DBX  580.3;
NETWORK
TITLE =#701 RBT1호 용접카운트 DATA CLEATR

      AN    M   1008.2;
      JNB   _012;
      L     0;
      T     DB42.DBW  420;
_012: NOP   0;
NETWORK
TITLE =#701 RBT2호 용접카운터 INT -> DB로 전송보조

      AN    OV;
      =     L      2.0;
      A     L      2.0;
      A     I   1044.0;
      =     M     12.0;
      A     L      2.0;
      A     I   1044.1;
      =     M     12.1;
      A     L      2.0;
      A     I   1044.2;
      =     M     12.2;
      A     L      2.0;
      A     I   1044.3;
      =     M     12.3;
      A     L      2.0;
      A     I   1044.4;
      =     M     12.4;
      A     L      2.0;
      A     OV;
      =     M     12.5;
      =     M     12.6;
      =     M     12.7;
NETWORK
TITLE =#701 RBT2호 용접카운터 INT -> DB로 전송
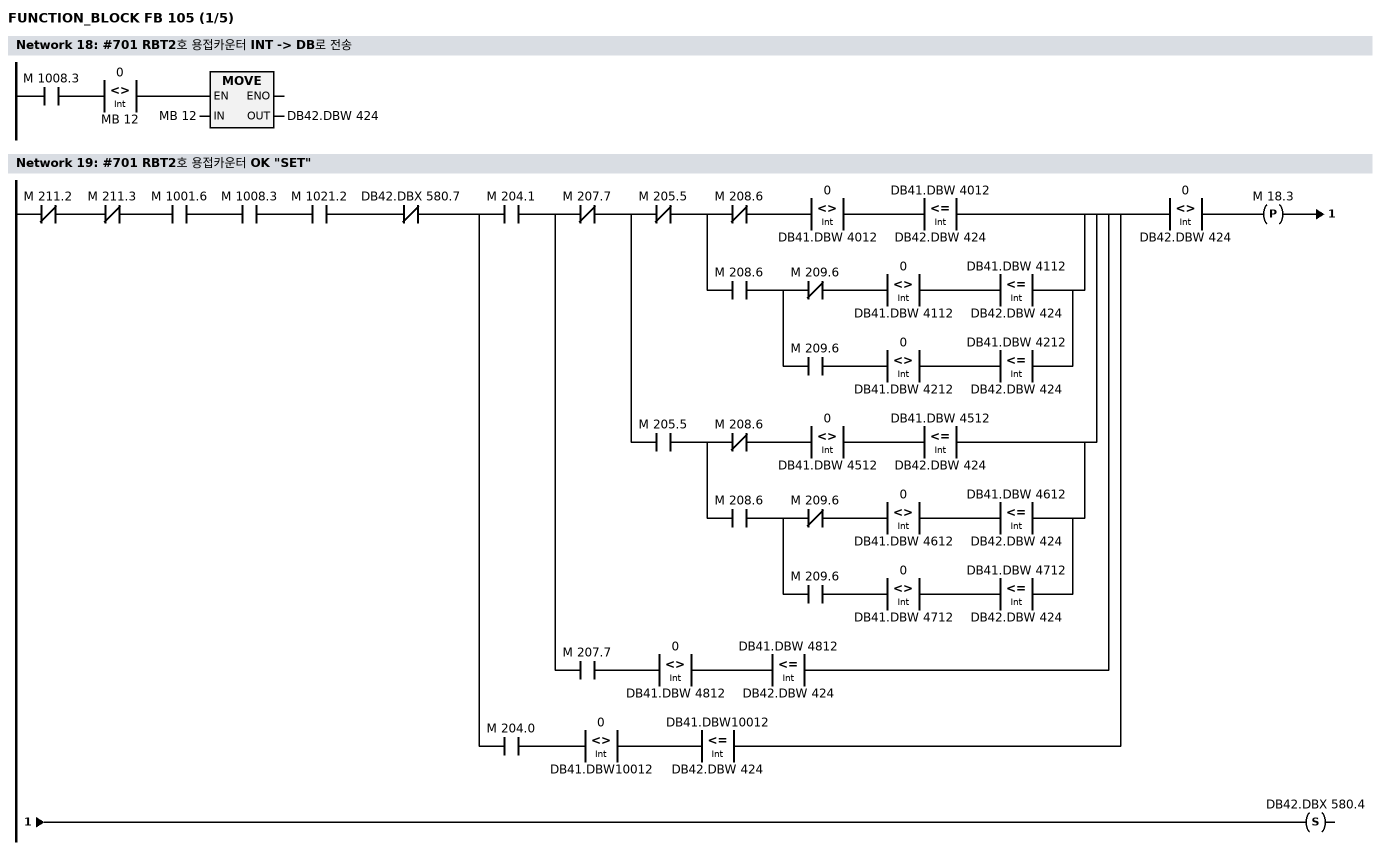

      A     M   1008.3;
      A(    ;
      L     0;
      L     MB    12;
      <>I   ;
      )     ;
      JNB   _013;
      L     MB    12;
      T     DB42.DBW  424;
_013: NOP   0;
NETWORK
TITLE =#701 RBT2호 용접카운터 OK "SET"

      AN    M    211.2;
      AN    M    211.3;
      A     M   1001.6;
      A     M   1008.3;
      A     M   1021.2;
      AN    DB42.DBX  580.7;
      A(    ;
      A     M    204.1;
      A(    ;
      AN    M    207.7;
      A(    ;
      AN    M    205.5;
      A(    ;
      AN    M    208.6;
      A(    ;
      L     0;
      L     DB41.DBW 4012;
      <>I   ;
      )     ;
      A(    ;
      L     DB41.DBW 4012;
      L     DB42.DBW  424;
      <=I   ;
      )     ;
      O     ;
      A     M    208.6;
      A(    ;
      AN    M    209.6;
      A(    ;
      L     0;
      L     DB41.DBW 4112;
      <>I   ;
      )     ;
      A(    ;
      L     DB41.DBW 4112;
      L     DB42.DBW  424;
      <=I   ;
      )     ;
      O     ;
      A     M    209.6;
      A(    ;
      L     0;
      L     DB41.DBW 4212;
      <>I   ;
      )     ;
      A(    ;
      L     DB41.DBW 4212;
      L     DB42.DBW  424;
      <=I   ;
      )     ;
      )     ;
      )     ;
      O     ;
      A     M    205.5;
      A(    ;
      AN    M    208.6;
      A(    ;
      L     0;
      L     DB41.DBW 4512;
      <>I   ;
      )     ;
      A(    ;
      L     DB41.DBW 4512;
      L     DB42.DBW  424;
      <=I   ;
      )     ;
      O     ;
      A     M    208.6;
      A(    ;
      AN    M    209.6;
      A(    ;
      L     0;
      L     DB41.DBW 4612;
      <>I   ;
      )     ;
      A(    ;
      L     DB41.DBW 4612;
      L     DB42.DBW  424;
      <=I   ;
      )     ;
      O     ;
      A     M    209.6;
      A(    ;
      L     0;
      L     DB41.DBW 4712;
      <>I   ;
      )     ;
      A(    ;
      L     DB41.DBW 4712;
      L     DB42.DBW  424;
      <=I   ;
      )     ;
      )     ;
      )     ;
      )     ;
      O     ;
      A     M    207.7;
      A(    ;
      L     0;
      L     DB41.DBW 4812;
      <>I   ;
      )     ;
      A(    ;
      L     DB41.DBW 4812;
      L     DB42.DBW  424;
      <=I   ;
      )     ;
      )     ;
      O     ;
      A     M    204.0;
      A(    ;
      L     0;
      L     DB41.DBW10012;
      <>I   ;
      )     ;
      A(    ;
      L     DB41.DBW10012;
      L     DB42.DBW  424;
      <=I   ;
      )     ;
      )     ;
      A(    ;
      L     0;
      L     DB42.DBW  424;
      <>I   ;
      )     ;
      FP    M     18.3;
      S     DB42.DBX  580.4;
NETWORK
TITLE =#701 RBT2호 용접카운터 NG "SET"
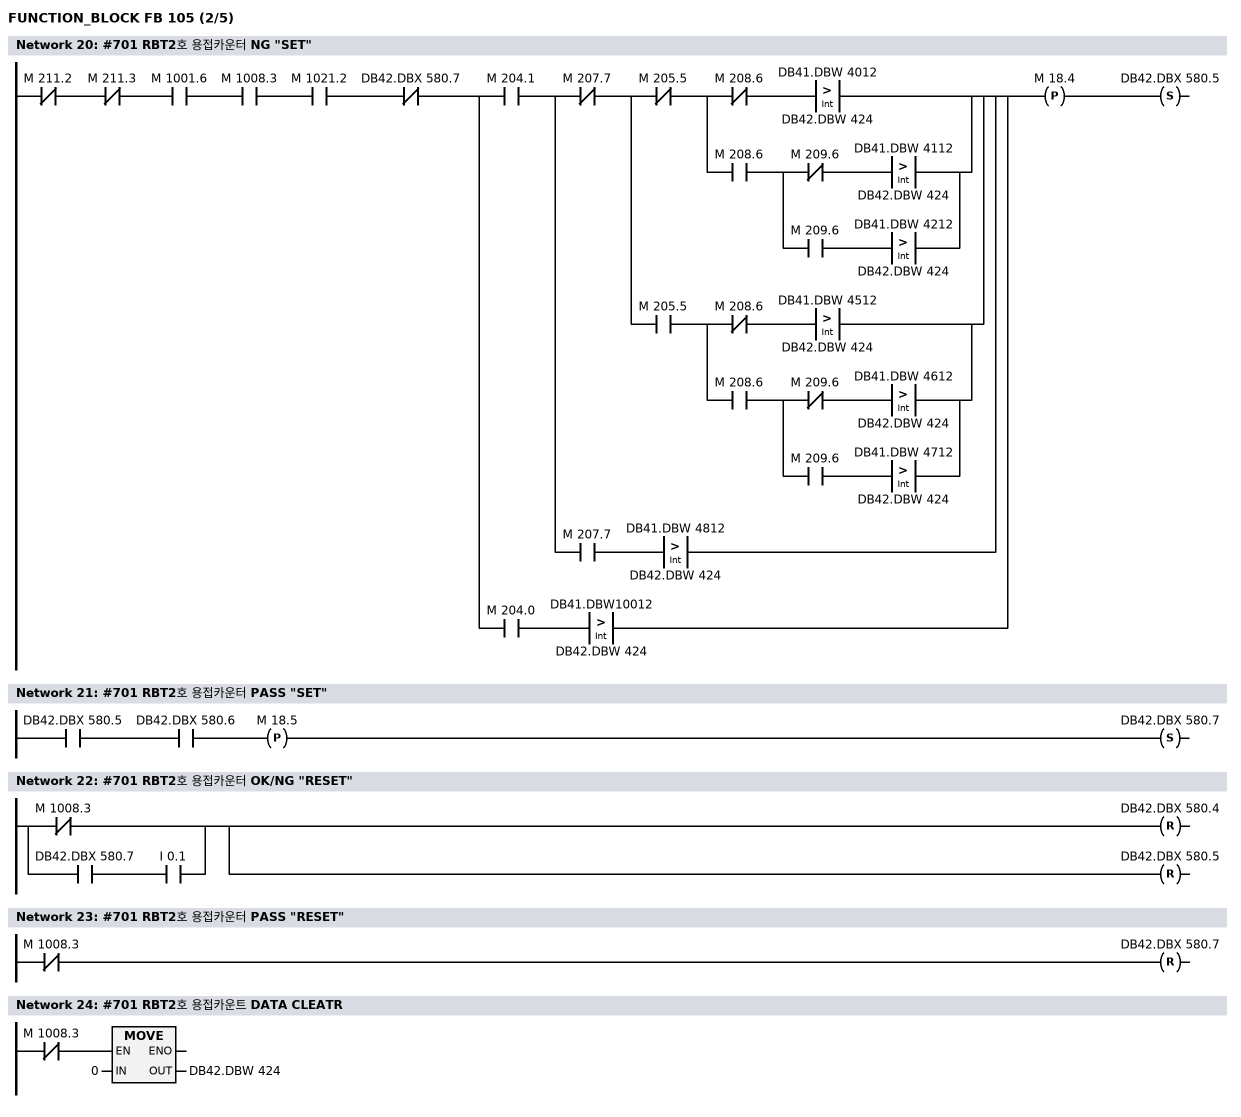

      AN    M    211.2;
      AN    M    211.3;
      A     M   1001.6;
      A     M   1008.3;
      A     M   1021.2;
      AN    DB42.DBX  580.7;
      A(    ;
      A     M    204.1;
      A(    ;
      AN    M    207.7;
      A(    ;
      AN    M    205.5;
      A(    ;
      AN    M    208.6;
      A(    ;
      L     DB41.DBW 4012;
      L     DB42.DBW  424;
      >I    ;
      )     ;
      O     ;
      A     M    208.6;
      A(    ;
      AN    M    209.6;
      A(    ;
      L     DB41.DBW 4112;
      L     DB42.DBW  424;
      >I    ;
      )     ;
      O     ;
      A     M    209.6;
      A(    ;
      L     DB41.DBW 4212;
      L     DB42.DBW  424;
      >I    ;
      )     ;
      )     ;
      )     ;
      O     ;
      A     M    205.5;
      A(    ;
      AN    M    208.6;
      A(    ;
      L     DB41.DBW 4512;
      L     DB42.DBW  424;
      >I    ;
      )     ;
      O     ;
      A     M    208.6;
      A(    ;
      AN    M    209.6;
      A(    ;
      L     DB41.DBW 4612;
      L     DB42.DBW  424;
      >I    ;
      )     ;
      O     ;
      A     M    209.6;
      A(    ;
      L     DB41.DBW 4712;
      L     DB42.DBW  424;
      >I    ;
      )     ;
      )     ;
      )     ;
      )     ;
      O     ;
      A     M    207.7;
      A(    ;
      L     DB41.DBW 4812;
      L     DB42.DBW  424;
      >I    ;
      )     ;
      )     ;
      O     ;
      A     M    204.0;
      A(    ;
      L     DB41.DBW10012;
      L     DB42.DBW  424;
      >I    ;
      )     ;
      )     ;
      FP    M     18.4;
      S     DB42.DBX  580.5;
NETWORK
TITLE =#701 RBT2호 용접카운터 PASS "SET"
//
//
      A     DB42.DBX  580.5;
      A     DB42.DBX  580.6;
      FP    M     18.5;
      S     DB42.DBX  580.7;
NETWORK
TITLE =#701 RBT2호 용접카운터 OK/NG "RESET"

      ON    M   1008.3;
      O     ;
      A     DB42.DBX  580.7;
      A     I      0.1;
      R     DB42.DBX  580.4;
      R     DB42.DBX  580.5;
NETWORK
TITLE =#701 RBT2호 용접카운터 PASS "RESET"

      AN    M   1008.3;
      R     DB42.DBX  580.7;
NETWORK
TITLE =#701 RBT2호 용접카운트 DATA CLEATR

      AN    M   1008.3;
      JNB   _014;
      L     0;
      T     DB42.DBW  424;
_014: NOP   0;
NETWORK
TITLE =#701 공정DATA
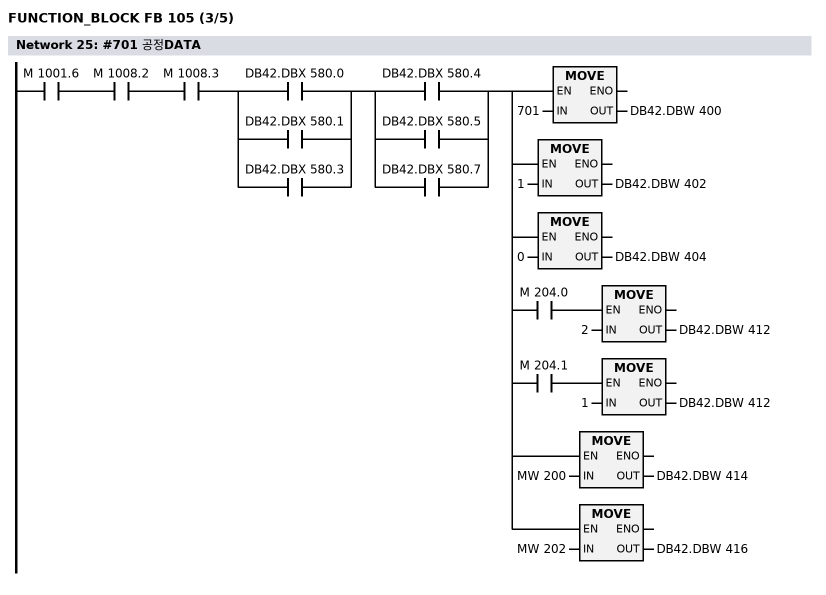

      A     M   1001.6;
      A     M   1008.2;
      A     M   1008.3;
      A(    ;
      O     DB42.DBX  580.0;
      O     DB42.DBX  580.1;
      O     DB42.DBX  580.3;
      )     ;
      A(    ;
      O     DB42.DBX  580.4;
      O     DB42.DBX  580.5;
      O     DB42.DBX  580.7;
      )     ;
      =     L      2.0;
      A     L      2.0;
      JNB   _015;
      L     701;
      T     DB42.DBW  400;
_015: NOP   0;
      A     L      2.0;
      JNB   _016;
      L     1;
      T     DB42.DBW  402;
_016: NOP   0;
      A     L      2.0;
      JNB   _017;
      L     0;
      T     DB42.DBW  404;
_017: NOP   0;
      A     L      2.0;
      A     M    204.0;
      JNB   _018;
      L     2;
      T     DB42.DBW  412;
_018: NOP   0;
      A     L      2.0;
      A     M    204.1;
      JNB   _019;
      L     1;
      T     DB42.DBW  412;
_019: NOP   0;
      A     L      2.0;
      JNB   _01a;
      L     MW   200;
      T     DB42.DBW  414;
_01a: NOP   0;
      A     L      2.0;
      JNB   _01b;
      L     MW   202;
      T     DB42.DBW  416;
_01b: NOP   0;
NETWORK
TITLE =#701R1,R2 CODE DATA
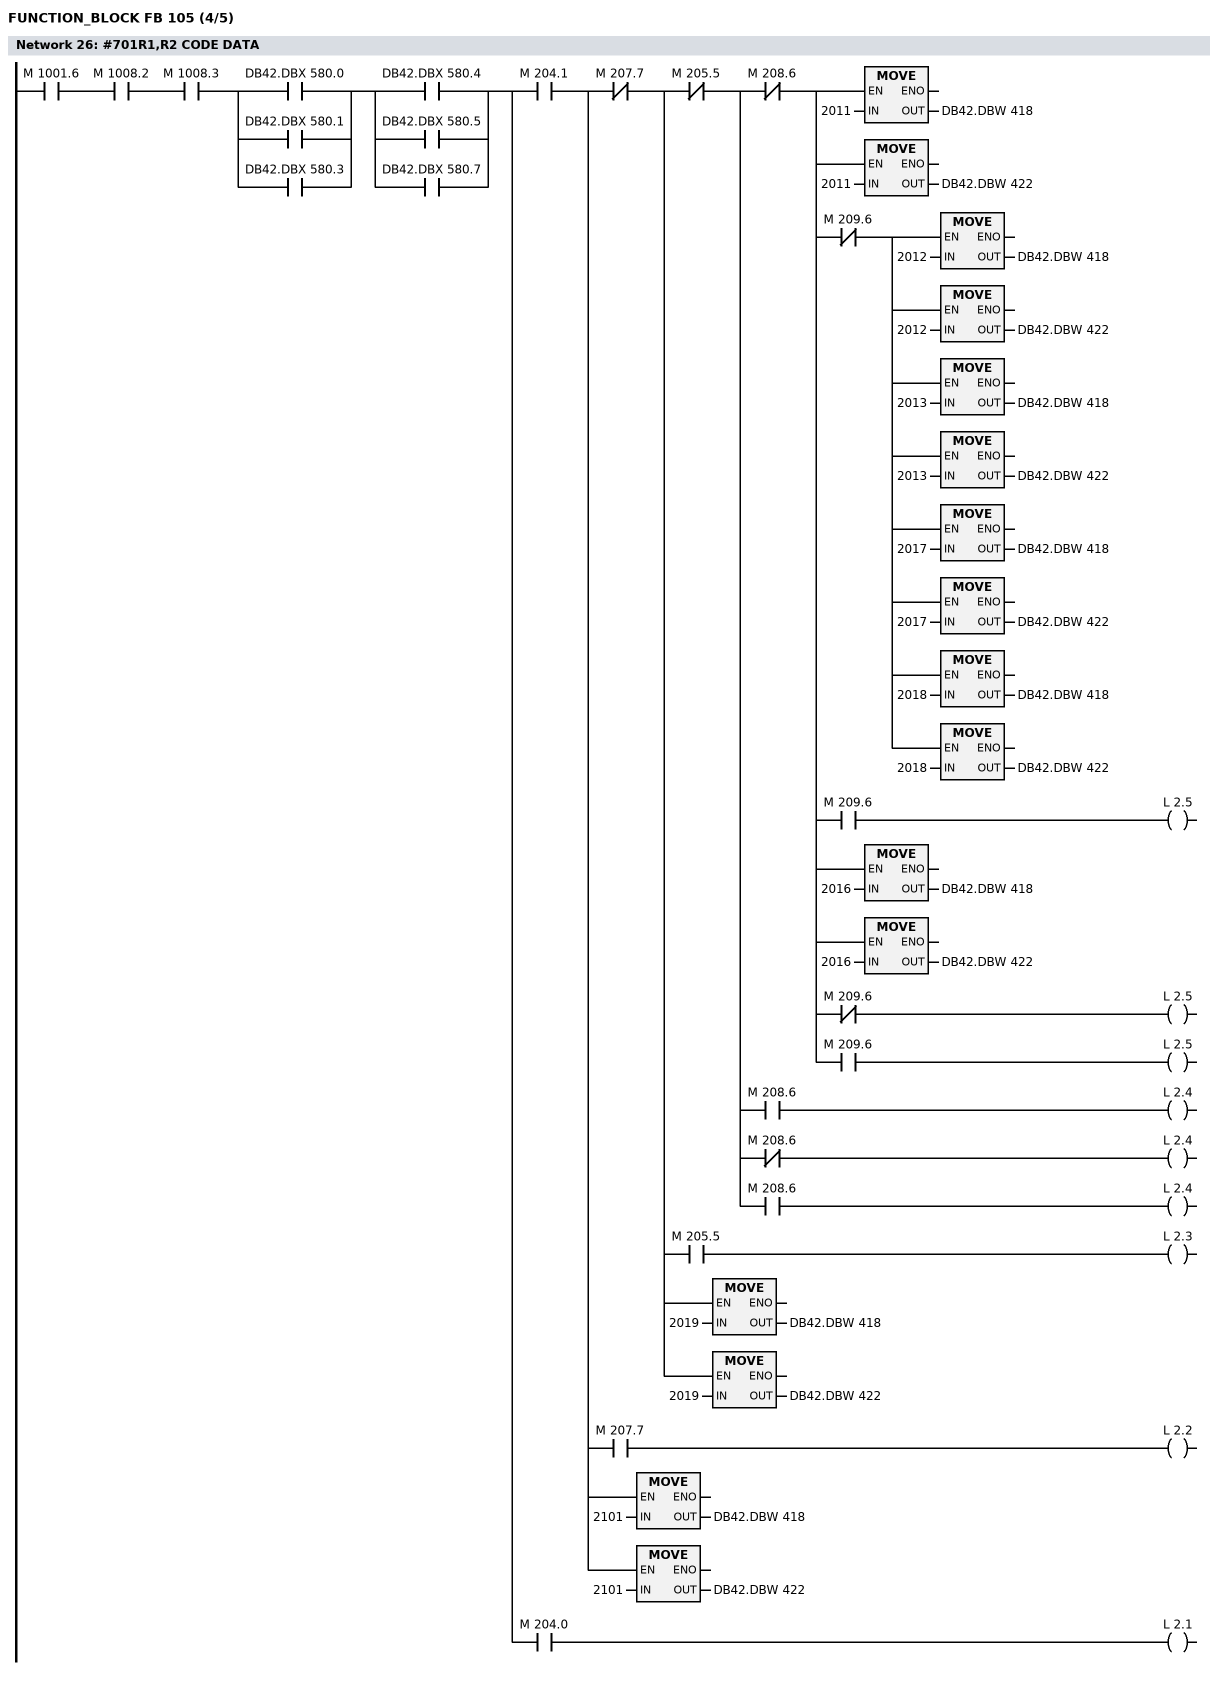

      A     M   1001.6;
      A     M   1008.2;
      A     M   1008.3;
      A(    ;
      O     DB42.DBX  580.0;
      O     DB42.DBX  580.1;
      O     DB42.DBX  580.3;
      )     ;
      A(    ;
      O     DB42.DBX  580.4;
      O     DB42.DBX  580.5;
      O     DB42.DBX  580.7;
      )     ;
      =     L      2.0;
      A     L      2.0;
      A     M    204.1;
      =     L      2.1;
      A     L      2.1;
      AN    M    207.7;
      =     L      2.2;
      A     L      2.2;
      AN    M    205.5;
      =     L      2.3;
      A     L      2.3;
      AN    M    208.6;
      =     L      2.4;
      A     L      2.4;
      JNB   _01c;
      L     2011;
      T     DB42.DBW  418;
_01c: NOP   0;
      A     L      2.4;
      JNB   _01d;
      L     2011;
      T     DB42.DBW  422;
_01d: NOP   0;
      A     L      2.3;
      A     M    208.6;
      =     L      2.4;
      A     L      2.4;
      AN    M    209.6;
      =     L      2.5;
      A     L      2.5;
      JNB   _01e;
      L     2012;
      T     DB42.DBW  418;
_01e: NOP   0;
      A     L      2.5;
      JNB   _01f;
      L     2012;
      T     DB42.DBW  422;
_01f: NOP   0;
      A     L      2.4;
      A     M    209.6;
      =     L      2.5;
      A     L      2.5;
      JNB   _020;
      L     2013;
      T     DB42.DBW  418;
_020: NOP   0;
      A     L      2.5;
      JNB   _021;
      L     2013;
      T     DB42.DBW  422;
_021: NOP   0;
      A     L      2.2;
      A     M    205.5;
      =     L      2.3;
      A     L      2.3;
      AN    M    208.6;
      =     L      2.4;
      A     L      2.4;
      JNB   _022;
      L     2016;
      T     DB42.DBW  418;
_022: NOP   0;
      A     L      2.4;
      JNB   _023;
      L     2016;
      T     DB42.DBW  422;
_023: NOP   0;
      A     L      2.3;
      A     M    208.6;
      =     L      2.4;
      A     L      2.4;
      AN    M    209.6;
      =     L      2.5;
      A     L      2.5;
      JNB   _024;
      L     2017;
      T     DB42.DBW  418;
_024: NOP   0;
      A     L      2.5;
      JNB   _025;
      L     2017;
      T     DB42.DBW  422;
_025: NOP   0;
      A     L      2.4;
      A     M    209.6;
      =     L      2.5;
      A     L      2.5;
      JNB   _026;
      L     2018;
      T     DB42.DBW  418;
_026: NOP   0;
      A     L      2.5;
      JNB   _027;
      L     2018;
      T     DB42.DBW  422;
_027: NOP   0;
      A     L      2.1;
      A     M    207.7;
      =     L      2.2;
      A     L      2.2;
      JNB   _028;
      L     2019;
      T     DB42.DBW  418;
_028: NOP   0;
      A     L      2.2;
      JNB   _029;
      L     2019;
      T     DB42.DBW  422;
_029: NOP   0;
      A     L      2.0;
      A     M    204.0;
      =     L      2.1;
      A     L      2.1;
      JNB   _02a;
      L     2101;
      T     DB42.DBW  418;
_02a: NOP   0;
      A     L      2.1;
      JNB   _02b;
      L     2101;
      T     DB42.DBW  422;
_02b: NOP   0;
NETWORK
TITLE =#701 용접결과
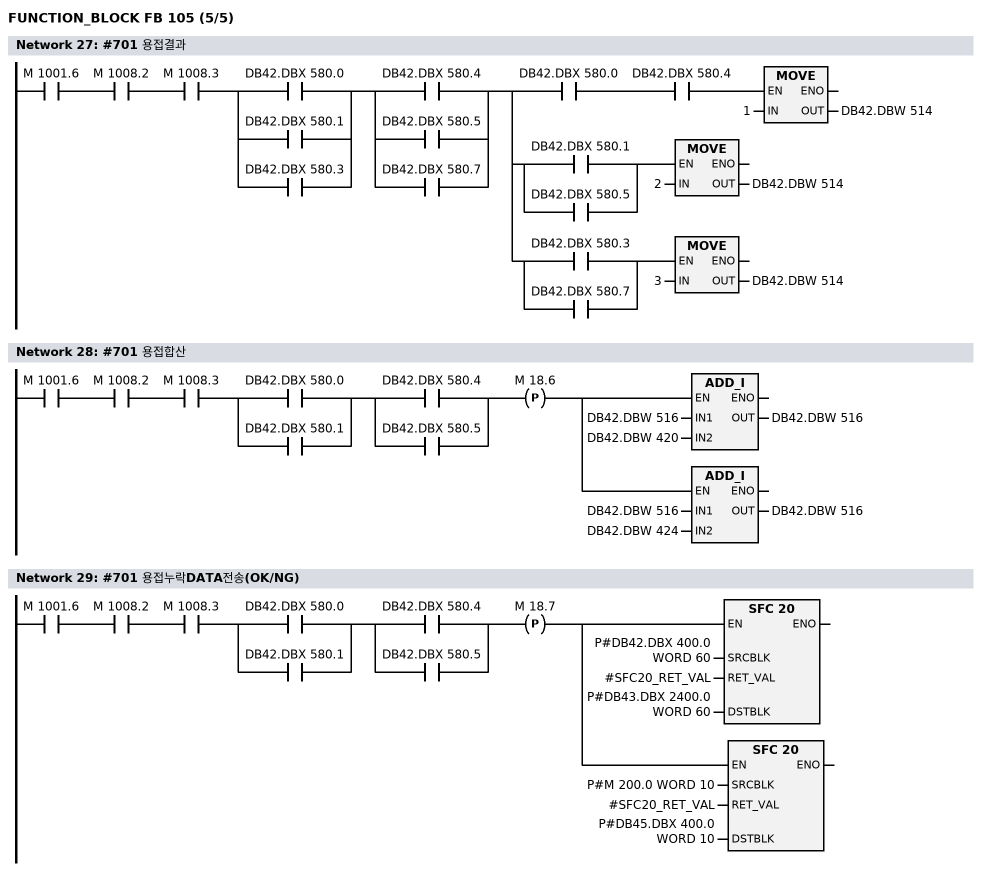

      A     M   1001.6;
      A     M   1008.2;
      A     M   1008.3;
      A(    ;
      O     DB42.DBX  580.0;
      O     DB42.DBX  580.1;
      O     DB42.DBX  580.3;
      )     ;
      A(    ;
      O     DB42.DBX  580.4;
      O     DB42.DBX  580.5;
      O     DB42.DBX  580.7;
      )     ;
      =     L      2.0;
      A     L      2.0;
      A     DB42.DBX  580.0;
      A     DB42.DBX  580.4;
      JNB   _02c;
      L     1;
      T     DB42.DBW  514;
_02c: NOP   0;
      A     L      2.0;
      A(    ;
      O     DB42.DBX  580.1;
      O     DB42.DBX  580.5;
      )     ;
      JNB   _02d;
      L     2;
      T     DB42.DBW  514;
_02d: NOP   0;
      A     L      2.0;
      A(    ;
      O     DB42.DBX  580.3;
      O     DB42.DBX  580.7;
      )     ;
      JNB   _02e;
      L     3;
      T     DB42.DBW  514;
_02e: NOP   0;
NETWORK
TITLE =#701 용접합산

      A     M   1001.6;
      A     M   1008.2;
      A     M   1008.3;
      A(    ;
      O     DB42.DBX  580.0;
      O     DB42.DBX  580.1;
      )     ;
      A(    ;
      O     DB42.DBX  580.4;
      O     DB42.DBX  580.5;
      )     ;
      FP    M     18.6;
      =     L      2.0;
      A     L      2.0;
      JNB   _02f;
      L     DB42.DBW  516;
      L     DB42.DBW  420;
      +I    ;
      T     DB42.DBW  516;
_02f: NOP   0;
      A     L      2.0;
      JNB   _030;
      L     DB42.DBW  516;
      L     DB42.DBW  424;
      +I    ;
      T     DB42.DBW  516;
_030: NOP   0;
NETWORK
TITLE =#701 용접누락DATA전송(OK/NG)

      A     M   1001.6;
      A     M   1008.2;
      A     M   1008.3;
      A(    ;
      O     DB42.DBX  580.0;
      O     DB42.DBX  580.1;
      )     ;
      A(    ;
      O     DB42.DBX  580.4;
      O     DB42.DBX  580.5;
      )     ;
      FP    M     18.7;
      =     L      2.0;
      A     L      2.0;
      JNB   _031;
      CALL SFC   20 (
           SRCBLK                   := P#DB42.DBX 400.0 WORD 60,
           RET_VAL                  := #SFC20_RET_VAL,
           DSTBLK                   := P#DB43.DBX 2400.0 WORD 60);
_031: NOP   0;
      A     L      2.0;
      JNB   _032;
      CALL SFC   20 (
           SRCBLK                   := P#M 200.0 WORD 10,
           RET_VAL                  := #SFC20_RET_VAL,
           DSTBLK                   := P#DB45.DBX 400.0 WORD 10);
_032: NOP   0;
NETWORK
TITLE =#701 용접누락BUFF전송

      A     M   1025.0;
      FP    M     19.0;
      =     L      2.0;
      A(    ;
      A     L      2.0;
      JNB   _033;
      CALL SFC   20 (
           SRCBLK                   := P#DB43.DBX 3360.0 WORD 60,
           RET_VAL                  := #SFC20_RET_VAL,
           DSTBLK                   := P#DB43.DBX 3480.0 WORD 60);
_033: A     BR;
      )     ;
      JNB   _034;
      CALL SFC   20 (
           SRCBLK                   := P#DB43.DBX 3240.0 WORD 60,
           RET_VAL                  := #SFC20_RET_VAL,
           DSTBLK                   := P#DB43.DBX 3360.0 WORD 60);
_034: NOP   0;
      A(    ;
      A     L      2.0;
      JNB   _035;
      CALL SFC   20 (
           SRCBLK                   := P#DB43.DBX 3120.0 WORD 60,
           RET_VAL                  := #SFC20_RET_VAL,
           DSTBLK                   := P#DB43.DBX 3240.0 WORD 60);
_035: A     BR;
      )     ;
      JNB   _036;
      CALL SFC   20 (
           SRCBLK                   := P#DB43.DBX 3000.0 WORD 60,
           RET_VAL                  := #SFC20_RET_VAL,
           DSTBLK                   := P#DB43.DBX 3120.0 WORD 60);
_036: NOP   0;
      A(    ;
      A     L      2.0;
      JNB   _037;
      CALL SFC   20 (
           SRCBLK                   := P#DB43.DBX 2880.0 WORD 60,
           RET_VAL                  := #SFC20_RET_VAL,
           DSTBLK                   := P#DB43.DBX 3000.0 WORD 60);
_037: A     BR;
      )     ;
      JNB   _038;
      CALL SFC   20 (
           SRCBLK                   := P#DB43.DBX 2760.0 WORD 60,
           RET_VAL                  := #SFC20_RET_VAL,
           DSTBLK                   := P#DB43.DBX 2880.0 WORD 60);
_038: NOP   0;
      A(    ;
      A     L      2.0;
      JNB   _039;
      CALL SFC   20 (
           SRCBLK                   := P#DB43.DBX 2640.0 WORD 60,
           RET_VAL                  := #SFC20_RET_VAL,
           DSTBLK                   := P#DB43.DBX 2760.0 WORD 60);
_039: A     BR;
      )     ;
      JNB   _03a;
      CALL SFC   20 (
           SRCBLK                   := P#DB43.DBX 2520.0 WORD 60,
           RET_VAL                  := #SFC20_RET_VAL,
           DSTBLK                   := P#DB43.DBX 2640.0 WORD 60);
_03a: NOP   0;
      A     L      2.0;
      JNB   _03b;
      CALL SFC   20 (
           SRCBLK                   := P#DB43.DBX 2400.0 WORD 60,
           RET_VAL                  := #SFC20_RET_VAL,
           DSTBLK                   := P#DB43.DBX 2520.0 WORD 60);
_03b: NOP   0;
      A     L      2.0;
      JNB   _03c;
      CALL SFC   21 (
           IN0                      := P#M 40.0 WORD 1,
           RET_VAL                  := #SFC20_RET_VAL,
           OUT1                     := P#DB43.DBX 2400.0 WORD 60);
_03c: NOP   0;
      A(    ;
      A     L      2.0;
      JNB   _03d;
      CALL SFC   20 (
           SRCBLK                   := P#DB45.DBX 560.0 WORD 10,
           RET_VAL                  := #SFC20_RET_VAL,
           DSTBLK                   := P#DB45.DBX 580.0 WORD 10);
_03d: A     BR;
      )     ;
      JNB   _03e;
      CALL SFC   20 (
           SRCBLK                   := P#DB45.DBX 540.0 WORD 10,
           RET_VAL                  := #SFC20_RET_VAL,
           DSTBLK                   := P#DB45.DBX 560.0 WORD 10);
_03e: NOP   0;
      A(    ;
      A     L      2.0;
      JNB   _03f;
      CALL SFC   20 (
           SRCBLK                   := P#DB45.DBX 520.0 WORD 10,
           RET_VAL                  := #SFC20_RET_VAL,
           DSTBLK                   := P#DB45.DBX 540.0 WORD 10);
_03f: A     BR;
      )     ;
      JNB   _040;
      CALL SFC   20 (
           SRCBLK                   := P#DB45.DBX 500.0 WORD 10,
           RET_VAL                  := #SFC20_RET_VAL,
           DSTBLK                   := P#DB45.DBX 520.0 WORD 10);
_040: NOP   0;
      A(    ;
      A     L      2.0;
      JNB   _041;
      CALL SFC   20 (
           SRCBLK                   := P#DB45.DBX 480.0 WORD 10,
           RET_VAL                  := #SFC20_RET_VAL,
           DSTBLK                   := P#DB45.DBX 500.0 WORD 10);
_041: A     BR;
      )     ;
      JNB   _042;
      CALL SFC   20 (
           SRCBLK                   := P#DB45.DBX 460.0 WORD 10,
           RET_VAL                  := #SFC20_RET_VAL,
           DSTBLK                   := P#DB45.DBX 480.0 WORD 10);
_042: NOP   0;
      A(    ;
      A     L      2.0;
      JNB   _043;
      CALL SFC   20 (
           SRCBLK                   := P#DB45.DBX 440.0 WORD 10,
           RET_VAL                  := #SFC20_RET_VAL,
           DSTBLK                   := P#DB45.DBX 460.0 WORD 10);
_043: A     BR;
      )     ;
      JNB   _044;
      CALL SFC   20 (
           SRCBLK                   := P#DB45.DBX 420.0 WORD 10,
           RET_VAL                  := #SFC20_RET_VAL,
           DSTBLK                   := P#DB45.DBX 440.0 WORD 10);
_044: NOP   0;
      A     L      2.0;
      JNB   _045;
      CALL SFC   20 (
           SRCBLK                   := P#DB45.DBX 400.0 WORD 10,
           RET_VAL                  := #SFC20_RET_VAL,
           DSTBLK                   := P#DB45.DBX 420.0 WORD 10);
_045: NOP   0;
      A     L      2.0;
      JNB   _046;
      CALL SFC   21 (
           IN0                      := P#M 40.0 WORD 1,
           RET_VAL                  := #SFC20_RET_VAL,
           OUT1                     := P#DB45.DBX 400.0 WORD 10);
_046: NOP   0;
NETWORK
TITLE =#701 용접누락DATA전송(PASS)
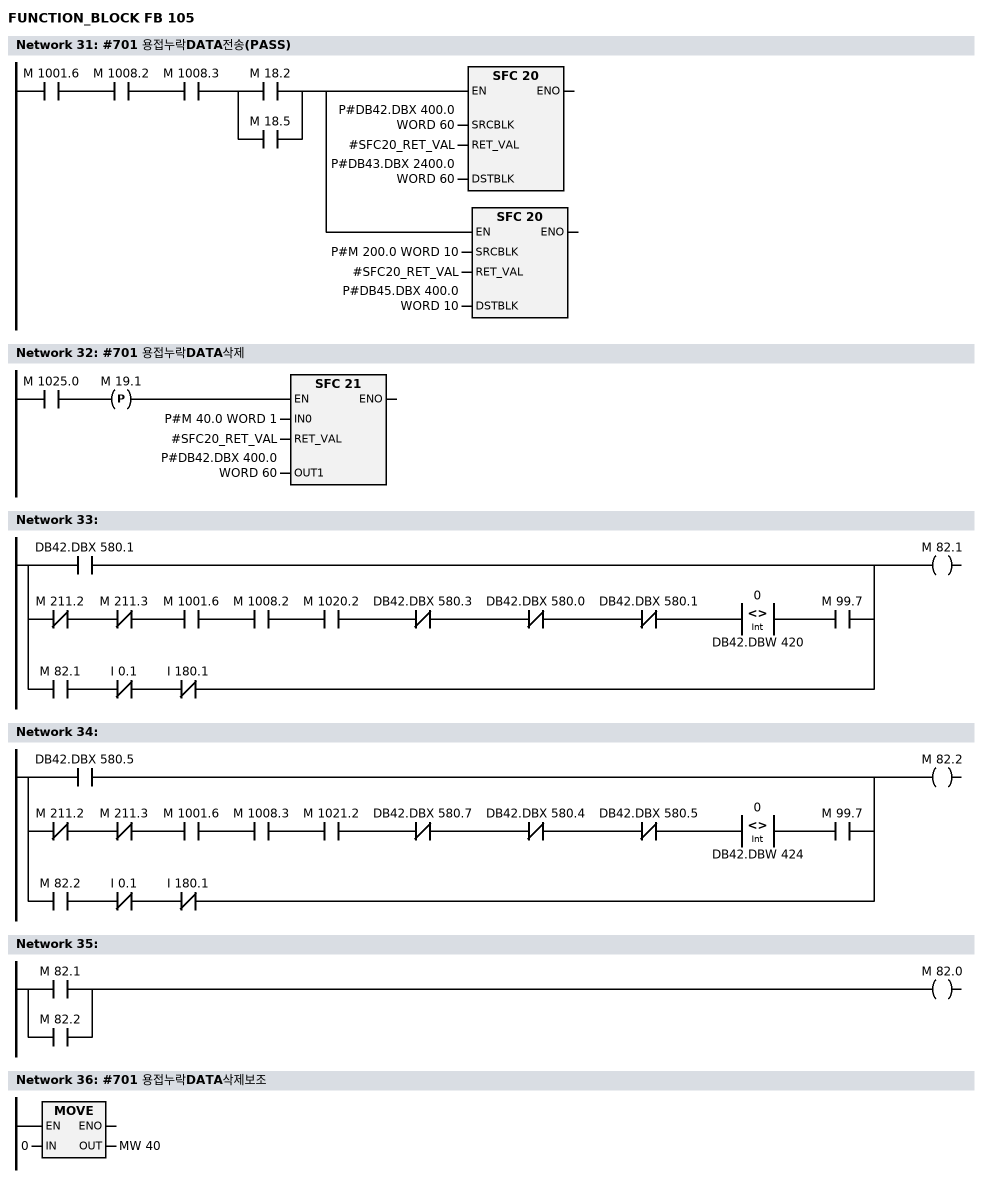

      A     M   1001.6;
      A     M   1008.2;
      A     M   1008.3;
      A(    ;
      O     M     18.2;
      O     M     18.5;
      )     ;
      =     L      2.0;
      A     L      2.0;
      JNB   _047;
      CALL SFC   20 (
           SRCBLK                   := P#DB42.DBX 400.0 WORD 60,
           RET_VAL                  := #SFC20_RET_VAL,
           DSTBLK                   := P#DB43.DBX 2400.0 WORD 60);
_047: NOP   0;
      A     L      2.0;
      JNB   _048;
      CALL SFC   20 (
           SRCBLK                   := P#M 200.0 WORD 10,
           RET_VAL                  := #SFC20_RET_VAL,
           DSTBLK                   := P#DB45.DBX 400.0 WORD 10);
_048: NOP   0;
NETWORK
TITLE =#701 용접누락DATA삭제

      A     M   1025.0;
      FP    M     19.1;
      JNB   _049;
      CALL SFC   21 (
           IN0                      := P#M 40.0 WORD 1,
           RET_VAL                  := #SFC20_RET_VAL,
           OUT1                     := P#DB42.DBX 400.0 WORD 60);
_049: NOP   0;
NETWORK
TITLE =

      O     DB42.DBX  580.1;
      O     ;
      AN    M    211.2;
      AN    M    211.3;
      A     M   1001.6;
      A     M   1008.2;
      A     M   1020.2;
      AN    DB42.DBX  580.3;
      AN    DB42.DBX  580.0;
      AN    DB42.DBX  580.1;
      A(    ;
      L     0;
      L     DB42.DBW  420;
      <>I   ;
      )     ;
      A     M     99.7;
      O     ;
      A     M     82.1;
      AN    I      0.1;
      AN    I    180.1;
      =     M     82.1;
NETWORK
TITLE =

      O     DB42.DBX  580.5;
      O     ;
      AN    M    211.2;
      AN    M    211.3;
      A     M   1001.6;
      A     M   1008.3;
      A     M   1021.2;
      AN    DB42.DBX  580.7;
      AN    DB42.DBX  580.4;
      AN    DB42.DBX  580.5;
      A(    ;
      L     0;
      L     DB42.DBW  424;
      <>I   ;
      )     ;
      A     M     99.7;
      O     ;
      A     M     82.2;
      AN    I      0.1;
      AN    I    180.1;
      =     M     82.2;
NETWORK
TITLE =

      O     M     82.1;
      O     M     82.2;
      =     M     82.0;
NETWORK
TITLE =#701 용접누락DATA삭제보조

      L     0;
      T     MW    40;
      NOP   0;
END_FUNCTION_BLOCK

DATA_BLOCK DB 105
TITLE =
VERSION : 0.0

 FB 105
BEGIN
   MW_0_BUFF[0] := W#16#0;
   MW_0_BUFF[1] := W#16#0;
   MW_0_BUFF[2] := W#16#0;
   MW_0_BUFF[3] := W#16#0;
   MW_0_BUFF[4] := W#16#0;
   MW_0_BUFF[5] := W#16#0;
   MW_0_BUFF[6] := W#16#0;
   MW_0_BUFF[7] := W#16#0;
   MW_0_BUFF[8] := W#16#0;
   MW_0_BUFF[9] := W#16#0;
   MW_0_BUFF[10] := W#16#0;
   MW_0_BUFF[11] := W#16#0;
   MW_0_BUFF[12] := W#16#0;
   MW_0_BUFF[13] := W#16#0;
   MW_0_BUFF[14] := W#16#0;
   MW_0_BUFF[15] := W#16#0;
   MW_0_BUFF[16] := W#16#0;
   MW_0_BUFF[17] := W#16#0;
   MW_0_BUFF[18] := W#16#0;
   MW_0_BUFF[19] := W#16#0;
   MW_0_BUFF[20] := W#16#0;
   MW_0_BUFF[21] := W#16#0;
   MW_0_BUFF[22] := W#16#0;
   MW_0_BUFF[23] := W#16#0;
   MW_0_BUFF[24] := W#16#0;
   MW_0_BUFF[25] := W#16#0;
   MW_0_BUFF[26] := W#16#0;
   MW_0_BUFF[27] := W#16#0;
   MW_0_BUFF[28] := W#16#0;
   MW_0_BUFF[29] := W#16#0;
   MW_0_BUFF[30] := W#16#0;
   MW_0_BUFF[31] := W#16#0;
   MW_0_BUFF[32] := W#16#0;
   MW_0_BUFF[33] := W#16#0;
   MW_0_BUFF[34] := W#16#0;
   MW_0_BUFF[35] := W#16#0;
   MW_0_BUFF[36] := W#16#0;
   MW_0_BUFF[37] := W#16#0;
   MW_0_BUFF[38] := W#16#0;
   MW_0_BUFF[39] := W#16#0;
   MW_0_BUFF[40] := W#16#0;
   MW_0_BUFF[41] := W#16#0;
   MW_0_BUFF[42] := W#16#0;
   MW_0_BUFF[43] := W#16#0;
   MW_0_BUFF[44] := W#16#0;
   MW_0_BUFF[45] := W#16#0;
   MW_0_BUFF[46] := W#16#0;
   MW_0_BUFF[47] := W#16#0;
   MW_0_BUFF[48] := W#16#0;
   MW_0_BUFF[49] := W#16#0;
   MW_0_BUFF[50] := W#16#0;
   MW_0_BUFF[51] := W#16#0;
   MW_0_BUFF[52] := W#16#0;
   MW_0_BUFF[53] := W#16#0;
   MW_0_BUFF[54] := W#16#0;
   MW_0_BUFF[55] := W#16#0;
   MW_0_BUFF[56] := W#16#0;
   MW_0_BUFF[57] := W#16#0;
   MW_0_BUFF[58] := W#16#0;
   MW_0_BUFF[59] := W#16#0;
   S701_RBT1_WELD_OK_PLS := FALSE;
   S701_RBT1_WELD_NG_PLS := FALSE;
   S701_RBT1_WELD_PASS_PLS := FALSE;
   S701_RBT2_WELD_OK_PLS := FALSE;
   S701_RBT2_WELD_NG_PLS := FALSE;
   S701_RBT2_WELD_PASS_PLS := FALSE;
   S701_CHECK_SUM_PLS := FALSE;
   S701_WELD_DATA_MOV_BUFF := FALSE;
   PLS1 := FALSE;
   PLS2 := FALSE;
END_DATA_BLOCK

FUNCTION_BLOCK FB 107
TITLE =
VERSION : 0.1


VAR
  S700_R1_CT : FB 500;
  S700_IDLE_CT : FB 500;
  S700_R2_CT : FB 500;
  S700_1_IDLE_CT : FB 500;
  S701_R3_CT : FB 500;
  S701_CT : FB 500;
  S701_R4_CT : FB 500;
END_VAR
BEGIN
NETWORK
TITLE =
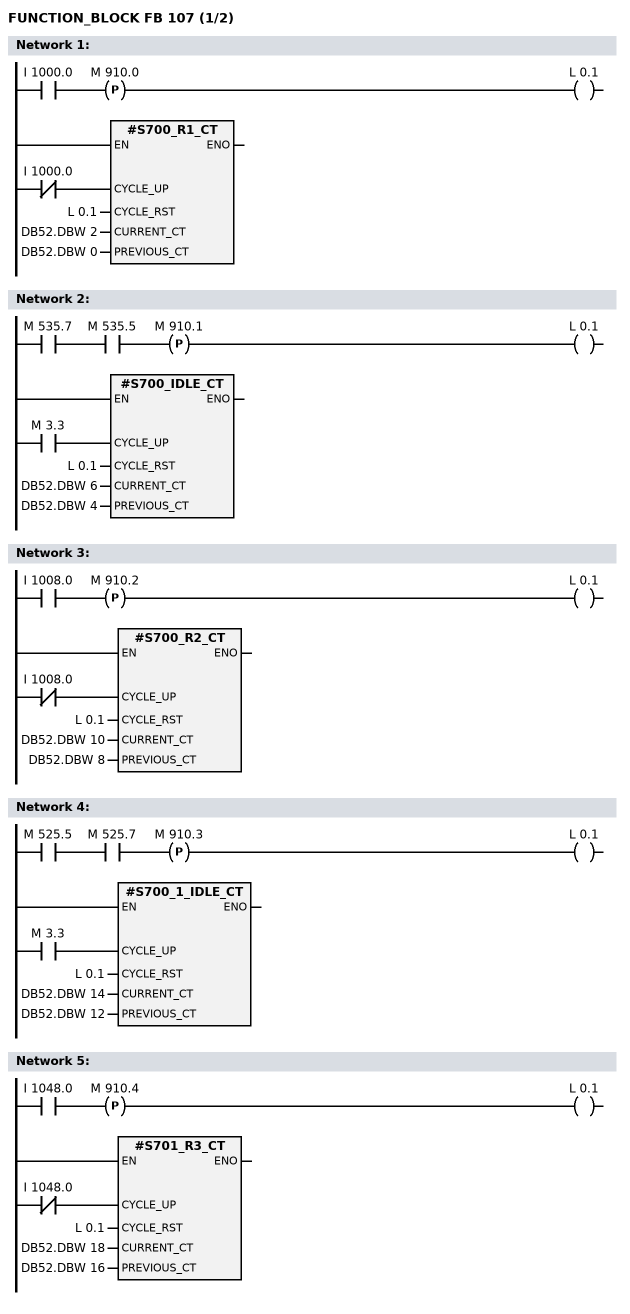

      AN    I   1000.0;
      =     L      0.0;
      BLD   103;
      A     I   1000.0;
      FP    M    910.0;
      =     L      0.1;
      BLD   103;
      CALL #S700_R1_CT (
           CYCLE_UP                 := L      0.0,
           CYCLE_RST                := L      0.1,
           CURRENT_CT               := DB52.DBW    2,
           PREVIOUS_CT              := DB52.DBW    0);
      NOP   0;
NETWORK
TITLE =

      A     M      3.3;
      =     L      0.0;
      BLD   103;
      A     M    535.7;
      A     M    535.5;
      FP    M    910.1;
      =     L      0.1;
      BLD   103;
      CALL #S700_IDLE_CT (
           CYCLE_UP                 := L      0.0,
           CYCLE_RST                := L      0.1,
           CURRENT_CT               := DB52.DBW    6,
           PREVIOUS_CT              := DB52.DBW    4);
      NOP   0;
NETWORK
TITLE =

      AN    I   1008.0;
      =     L      0.0;
      BLD   103;
      A     I   1008.0;
      FP    M    910.2;
      =     L      0.1;
      BLD   103;
      CALL #S700_R2_CT (
           CYCLE_UP                 := L      0.0,
           CYCLE_RST                := L      0.1,
           CURRENT_CT               := DB52.DBW   10,
           PREVIOUS_CT              := DB52.DBW    8);
      NOP   0;
NETWORK
TITLE =

      A     M      3.3;
      =     L      0.0;
      BLD   103;
      A     M    525.5;
      A     M    525.7;
      FP    M    910.3;
      =     L      0.1;
      BLD   103;
      CALL #S700_1_IDLE_CT (
           CYCLE_UP                 := L      0.0,
           CYCLE_RST                := L      0.1,
           CURRENT_CT               := DB52.DBW   14,
           PREVIOUS_CT              := DB52.DBW   12);
      NOP   0;
NETWORK
TITLE =

      AN    I   1048.0;
      =     L      0.0;
      BLD   103;
      A     I   1048.0;
      FP    M    910.4;
      =     L      0.1;
      BLD   103;
      CALL #S701_R3_CT (
           CYCLE_UP                 := L      0.0,
           CYCLE_RST                := L      0.1,
           CURRENT_CT               := DB52.DBW   18,
           PREVIOUS_CT              := DB52.DBW   16);
      NOP   0;
NETWORK
TITLE =
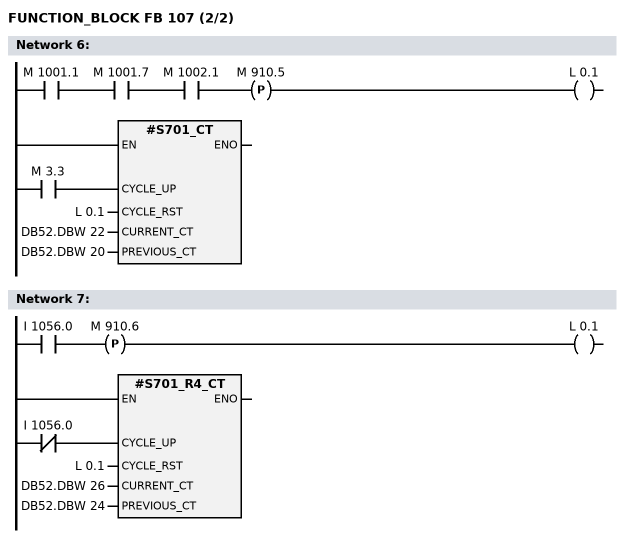

      A     M      3.3;
      =     L      0.0;
      BLD   103;
      A     M   1001.1;
      A     M   1001.7;
      A     M   1002.1;
      FP    M    910.5;
      =     L      0.1;
      BLD   103;
      CALL #S701_CT (
           CYCLE_UP                 := L      0.0,
           CYCLE_RST                := L      0.1,
           CURRENT_CT               := DB52.DBW   22,
           PREVIOUS_CT              := DB52.DBW   20);
      NOP   0;
NETWORK
TITLE =

      AN    I   1056.0;
      =     L      0.0;
      BLD   103;
      A     I   1056.0;
      FP    M    910.6;
      =     L      0.1;
      BLD   103;
      CALL #S701_R4_CT (
           CYCLE_UP                 := L      0.0,
           CYCLE_RST                := L      0.1,
           CURRENT_CT               := DB52.DBW   26,
           PREVIOUS_CT              := DB52.DBW   24);
      NOP   0;
END_FUNCTION_BLOCK

DATA_BLOCK DB 107
TITLE =
VERSION : 0.0

 FB 107
BEGIN
   S700_R1_CT.CYCLE_UP := FALSE;
   S700_R1_CT.CYCLE_RST := FALSE;
   S700_R1_CT.CURRENT_CT := 0;
   S700_R1_CT.PREVIOUS_CT := 0;
   S700_R1_CT.CURRENT := 0;
   S700_R1_CT.PREVIOUS := 0;
   S700_R1_CT.CYCLE_UP_PLS := FALSE;
   S700_R1_CT.CYCLE_RST_PLS := FALSE;
   S700_R1_CT.CYCLE_OVER_PLS := FALSE;
   S700_IDLE_CT.CYCLE_UP := FALSE;
   S700_IDLE_CT.CYCLE_RST := FALSE;
   S700_IDLE_CT.CURRENT_CT := 0;
   S700_IDLE_CT.PREVIOUS_CT := 0;
   S700_IDLE_CT.CURRENT := 0;
   S700_IDLE_CT.PREVIOUS := 0;
   S700_IDLE_CT.CYCLE_UP_PLS := FALSE;
   S700_IDLE_CT.CYCLE_RST_PLS := FALSE;
   S700_IDLE_CT.CYCLE_OVER_PLS := FALSE;
   S700_R2_CT.CYCLE_UP := FALSE;
   S700_R2_CT.CYCLE_RST := FALSE;
   S700_R2_CT.CURRENT_CT := 0;
   S700_R2_CT.PREVIOUS_CT := 0;
   S700_R2_CT.CURRENT := 0;
   S700_R2_CT.PREVIOUS := 0;
   S700_R2_CT.CYCLE_UP_PLS := FALSE;
   S700_R2_CT.CYCLE_RST_PLS := FALSE;
   S700_R2_CT.CYCLE_OVER_PLS := FALSE;
   S700_1_IDLE_CT.CYCLE_UP := FALSE;
   S700_1_IDLE_CT.CYCLE_RST := FALSE;
   S700_1_IDLE_CT.CURRENT_CT := 0;
   S700_1_IDLE_CT.PREVIOUS_CT := 0;
   S700_1_IDLE_CT.CURRENT := 0;
   S700_1_IDLE_CT.PREVIOUS := 0;
   S700_1_IDLE_CT.CYCLE_UP_PLS := FALSE;
   S700_1_IDLE_CT.CYCLE_RST_PLS := FALSE;
   S700_1_IDLE_CT.CYCLE_OVER_PLS := FALSE;
   S701_R3_CT.CYCLE_UP := FALSE;
   S701_R3_CT.CYCLE_RST := FALSE;
   S701_R3_CT.CURRENT_CT := 0;
   S701_R3_CT.PREVIOUS_CT := 0;
   S701_R3_CT.CURRENT := 0;
   S701_R3_CT.PREVIOUS := 0;
   S701_R3_CT.CYCLE_UP_PLS := FALSE;
   S701_R3_CT.CYCLE_RST_PLS := FALSE;
   S701_R3_CT.CYCLE_OVER_PLS := FALSE;
   S701_CT.CYCLE_UP := FALSE;
   S701_CT.CYCLE_RST := FALSE;
   S701_CT.CURRENT_CT := 0;
   S701_CT.PREVIOUS_CT := 0;
   S701_CT.CURRENT := 0;
   S701_CT.PREVIOUS := 0;
   S701_CT.CYCLE_UP_PLS := FALSE;
   S701_CT.CYCLE_RST_PLS := FALSE;
   S701_CT.CYCLE_OVER_PLS := FALSE;
   S701_R4_CT.CYCLE_UP := FALSE;
   S701_R4_CT.CYCLE_RST := FALSE;
   S701_R4_CT.CURRENT_CT := 0;
   S701_R4_CT.PREVIOUS_CT := 0;
   S701_R4_CT.CURRENT := 0;
   S701_R4_CT.PREVIOUS := 0;
   S701_R4_CT.CYCLE_UP_PLS := FALSE;
   S701_R4_CT.CYCLE_RST_PLS := FALSE;
   S701_R4_CT.CYCLE_OVER_PLS := FALSE;
END_DATA_BLOCK

FUNCTION_BLOCK FB 108
TITLE =
VERSION : 0.1

BEGIN
NETWORK
TITLE =PROFINET ERROR(1~10)
//
//
      A     M      3.3;
      =     L      0.0;
      A     L      0.0;
      A(    ;
      O     DB327.DBX 1025.3;
      O     ;
      A     M   7000.0;
      AN    I      0.1;
      AN    I    180.1;
      )     ;
      =     L      0.1;
      A     L      0.1;
      A     T    700;
      =     M   7000.0;
      A     L      0.1;
      BLD   102;
      L     S5T#0MS;
      SD    T    700;
      A     L      0.0;
      A(    ;
      O     DB327.DBX 1027.3;
      O     ;
      A     M   7000.1;
      AN    I      0.1;
      AN    I    180.1;
      )     ;
      =     L      0.1;
      A     L      0.1;
      A     T    701;
      =     M   7000.1;
      A     L      0.1;
      BLD   102;
      L     S5T#0MS;
      SD    T    701;
      A     L      0.0;
      A(    ;
      O     DB327.DBX 1029.3;
      O     ;
      A     M   7000.2;
      AN    I      0.1;
      AN    I    180.1;
      )     ;
      =     L      0.1;
      A     L      0.1;
      A     T    702;
      =     M   7000.2;
      A     L      0.1;
      BLD   102;
      L     S5T#0MS;
      SD    T    702;
      A     L      0.0;
      A(    ;
      O     DB327.DBX 1031.3;
      O     ;
      A     M   7000.3;
      AN    I      0.1;
      AN    I    180.1;
      )     ;
      =     L      0.1;
      A     L      0.1;
      A     T    703;
      =     M   7000.3;
      A     L      0.1;
      BLD   102;
      L     S5T#0MS;
      SD    T    703;
      A     L      0.0;
      A(    ;
      O     DB327.DBX 1033.3;
      O     ;
      A     M   7000.4;
      AN    I      0.1;
      AN    I    180.1;
      )     ;
      =     L      0.1;
      A     L      0.1;
      A     T    704;
      =     M   7000.4;
      A     L      0.1;
      BLD   102;
      L     S5T#0MS;
      SD    T    704;
      A     L      0.0;
      A(    ;
      O     DB327.DBX 1035.3;
      O     ;
      A     M   7000.5;
      AN    I      0.1;
      AN    I    180.1;
      )     ;
      =     L      0.1;
      A     L      0.1;
      A     T    705;
      =     M   7000.5;
      A     L      0.1;
      BLD   102;
      L     S5T#0MS;
      SD    T    705;
      A     L      0.0;
      A(    ;
      O     DB327.DBX 1037.3;
      O     ;
      A     M   7000.6;
      AN    I      0.1;
      AN    I    180.1;
      )     ;
      =     L      0.1;
      A     L      0.1;
      A     T    706;
      =     M   7000.6;
      A     L      0.1;
      BLD   102;
      L     S5T#0MS;
      SD    T    706;
      A     L      0.0;
      A(    ;
      O     DB327.DBX 1039.3;
      O     ;
      A     M   7000.7;
      AN    I      0.1;
      AN    I    180.1;
      )     ;
      =     L      0.1;
      A     L      0.1;
      A     T    707;
      =     M   7000.7;
      A     L      0.1;
      BLD   102;
      L     S5T#0MS;
      SD    T    707;
      A     L      0.0;
      A(    ;
      O     DB327.DBX 1041.3;
      O     ;
      A     M   7001.0;
      AN    I      0.1;
      AN    I    180.1;
      )     ;
      =     L      0.1;
      A     L      0.1;
      A     T    708;
      =     M   7001.0;
      A     L      0.1;
      BLD   102;
      L     S5T#0MS;
      SD    T    708;
      A     L      0.0;
      A(    ;
      O     DB327.DBX 1043.3;
      O     ;
      A     M   7001.1;
      AN    I      0.1;
      AN    I    180.1;
      )     ;
      =     L      0.1;
      A     L      0.1;
      A     T    709;
      =     M   7001.1;
      A     L      0.1;
      BLD   102;
      L     S5T#0MS;
      SD    T    709;
NETWORK
TITLE =PROFINET ERROR(11~20)
//
//
      A     M      3.3;
      =     L      0.0;
      A     L      0.0;
      A(    ;
      O     DB327.DBX 1045.3;
      O     ;
      A     M   7001.2;
      AN    I      0.1;
      AN    I    180.1;
      )     ;
      =     L      0.1;
      A     L      0.1;
      A     T    710;
      =     M   7001.2;
      A     L      0.1;
      BLD   102;
      L     S5T#0MS;
      SD    T    710;
      A     L      0.0;
      A(    ;
      O     DB327.DBX 1047.3;
      O     ;
      A     M   7001.3;
      AN    I      0.1;
      AN    I    180.1;
      )     ;
      =     L      0.1;
      A     L      0.1;
      A     T    711;
      =     M   7001.3;
      A     L      0.1;
      BLD   102;
      L     S5T#0MS;
      SD    T    711;
      A     L      0.0;
      A(    ;
      O     DB327.DBX 1049.3;
      O     ;
      A     M   7001.4;
      AN    I      0.1;
      AN    I    180.1;
      )     ;
      =     L      0.1;
      A     L      0.1;
      A     T    712;
      =     M   7001.4;
      A     L      0.1;
      BLD   102;
      L     S5T#0MS;
      SD    T    712;
      A     L      0.0;
      A(    ;
      O     DB327.DBX 1051.3;
      O     ;
      A     M   7001.5;
      AN    I      0.1;
      AN    I    180.1;
      )     ;
      =     L      0.1;
      A     L      0.1;
      A     T    713;
      =     M   7001.5;
      A     L      0.1;
      BLD   102;
      L     S5T#0MS;
      SD    T    713;
      A     L      0.0;
      A(    ;
      O     DB327.DBX 1053.3;
      O     ;
      A     M   7001.6;
      AN    I      0.1;
      AN    I    180.1;
      )     ;
      =     L      0.1;
      A     L      0.1;
      A     T    714;
      =     M   7001.6;
      A     L      0.1;
      BLD   102;
      L     S5T#0MS;
      SD    T    714;
      A     L      0.0;
      A(    ;
      O     DB327.DBX 1055.3;
      O     ;
      A     M   7001.7;
      AN    I      0.1;
      AN    I    180.1;
      )     ;
      =     L      0.1;
      A     L      0.1;
      A     T    715;
      =     M   7001.7;
      A     L      0.1;
      BLD   102;
      L     S5T#0MS;
      SD    T    715;
      A     L      0.0;
      A(    ;
      O     DB327.DBX 1057.3;
      O     ;
      A     M   7002.0;
      AN    I      0.1;
      AN    I    180.1;
      )     ;
      =     L      0.1;
      A     L      0.1;
      A     T    716;
      =     M   7002.0;
      A     L      0.1;
      BLD   102;
      L     S5T#0MS;
      SD    T    716;
      A     L      0.0;
      A(    ;
      O     DB327.DBX 1059.3;
      O     ;
      A     M   7002.1;
      AN    I      0.1;
      AN    I    180.1;
      )     ;
      =     L      0.1;
      A     L      0.1;
      A     T    717;
      =     M   7002.1;
      A     L      0.1;
      BLD   102;
      L     S5T#0MS;
      SD    T    717;
      A     L      0.0;
      A(    ;
      O     DB327.DBX 1061.3;
      O     ;
      A     M   7002.2;
      AN    I      0.1;
      AN    I    180.1;
      )     ;
      =     L      0.1;
      A     L      0.1;
      A     T    718;
      =     M   7002.2;
      A     L      0.1;
      BLD   102;
      L     S5T#0MS;
      SD    T    718;
      A     L      0.0;
      A(    ;
      O     DB327.DBX 1063.3;
      O     ;
      A     M   7002.3;
      AN    I      0.1;
      AN    I    180.1;
      )     ;
      =     L      0.1;
      A     L      0.1;
      A     T    719;
      =     M   7002.3;
      A     L      0.1;
      BLD   102;
      L     S5T#0MS;
      SD    T    719;
NETWORK
TITLE =PROFINET ERROR(21~30)
//
//
      A     M      3.3;
      =     L      0.0;
      A     L      0.0;
      A(    ;
      O     DB327.DBX 1065.3;
      O     ;
      A     M   7002.4;
      AN    I      0.1;
      AN    I    180.1;
      )     ;
      =     L      0.1;
      A     L      0.1;
      A     T    720;
      =     M   7002.4;
      A     L      0.1;
      BLD   102;
      L     S5T#0MS;
      SD    T    720;
      A     L      0.0;
      A(    ;
      O     DB327.DBX 1067.3;
      O     ;
      A     M   7002.5;
      AN    I      0.1;
      AN    I    180.1;
      )     ;
      =     L      0.1;
      A     L      0.1;
      A     T    721;
      =     M   7002.5;
      A     L      0.1;
      BLD   102;
      L     S5T#0MS;
      SD    T    721;
      A     L      0.0;
      A(    ;
      O     DB327.DBX 1069.3;
      O     ;
      A     M   7002.6;
      AN    I      0.1;
      AN    I    180.1;
      )     ;
      =     L      0.1;
      A     L      0.1;
      A     T    722;
      =     M   7002.6;
      A     L      0.1;
      BLD   102;
      L     S5T#0MS;
      SD    T    722;
      A     L      0.0;
      A(    ;
      O     DB327.DBX 1071.3;
      O     ;
      A     M   7002.7;
      AN    I      0.1;
      AN    I    180.1;
      )     ;
      =     L      0.1;
      A     L      0.1;
      A     T    723;
      =     M   7002.7;
      A     L      0.1;
      BLD   102;
      L     S5T#0MS;
      SD    T    723;
      A     L      0.0;
      A(    ;
      O     DB327.DBX 1073.3;
      O     ;
      A     M   7003.0;
      AN    I      0.1;
      AN    I    180.1;
      )     ;
      =     L      0.1;
      A     L      0.1;
      A     T    724;
      =     M   7003.0;
      A     L      0.1;
      BLD   102;
      L     S5T#0MS;
      SD    T    724;
      A     L      0.0;
      A(    ;
      O     DB327.DBX 1075.3;
      O     ;
      A     M   7003.1;
      AN    I      0.1;
      AN    I    180.1;
      )     ;
      =     L      0.1;
      A     L      0.1;
      A     T    725;
      =     M   7003.1;
      A     L      0.1;
      BLD   102;
      L     S5T#0MS;
      SD    T    725;
      A     L      0.0;
      A(    ;
      O     DB327.DBX 1077.3;
      O     ;
      A     M   7003.2;
      AN    I      0.1;
      AN    I    180.1;
      )     ;
      =     L      0.1;
      A     L      0.1;
      A     T    726;
      =     M   7003.2;
      A     L      0.1;
      BLD   102;
      L     S5T#0MS;
      SD    T    726;
      A     L      0.0;
      A(    ;
      O     DB327.DBX 1079.3;
      O     ;
      A     M   7003.3;
      AN    I      0.1;
      AN    I    180.1;
      )     ;
      =     L      0.1;
      A     L      0.1;
      A     T    727;
      AN    M      3.3;
      =     M   7003.3;
      A     L      0.1;
      BLD   102;
      L     S5T#0MS;
      SD    T    727;
      A     L      0.0;
      A(    ;
      O     DB327.DBX 1081.3;
      O     ;
      A     M   7003.4;
      AN    I      0.1;
      AN    I    180.1;
      )     ;
      =     L      0.1;
      A     L      0.1;
      A     T    728;
      AN    M      3.3;
      =     M   7003.4;
      A     L      0.1;
      BLD   102;
      L     S5T#0MS;
      SD    T    728;
      A     L      0.0;
      A(    ;
      O     DB327.DBX 1083.3;
      O     ;
      A     M   7003.5;
      AN    I      0.1;
      AN    I    180.1;
      )     ;
      =     L      0.1;
      A     L      0.1;
      A     T    729;
      AN    M      3.3;
      =     M   7003.5;
      A     L      0.1;
      BLD   102;
      L     S5T#0MS;
      SD    T    729;
NETWORK
TITLE =PROFINET ERROR(31~40)
//
//
      A     M      3.3;
      =     L      0.0;
      A     L      0.0;
      A(    ;
      O     DB327.DBX 1085.3;
      O     ;
      A     M   7003.6;
      AN    I      0.1;
      AN    I    180.1;
      )     ;
      =     L      0.1;
      A     L      0.1;
      A     T    730;
      AN    M      3.3;
      =     M   7003.6;
      A     L      0.1;
      BLD   102;
      L     S5T#0MS;
      SD    T    730;
      A     L      0.0;
      A(    ;
      O     DB327.DBX 1087.3;
      O     ;
      A     M   7003.7;
      AN    I      0.1;
      AN    I    180.1;
      )     ;
      =     L      0.1;
      A     L      0.1;
      A     T    731;
      AN    M      3.3;
      =     M   7003.7;
      A     L      0.1;
      BLD   102;
      L     S5T#0MS;
      SD    T    731;
      A     L      0.0;
      A(    ;
      O     DB327.DBX 1089.3;
      O     ;
      A     M   7004.0;
      AN    I      0.1;
      AN    I    180.1;
      )     ;
      =     L      0.1;
      A     L      0.1;
      A     T    732;
      AN    M      3.3;
      =     M   7004.0;
      A     L      0.1;
      BLD   102;
      L     S5T#0MS;
      SD    T    732;
      A     L      0.0;
      A(    ;
      O     DB327.DBX 1091.3;
      O     ;
      A     M   7004.1;
      AN    I      0.1;
      AN    I    180.1;
      )     ;
      =     L      0.1;
      A     L      0.1;
      A     T    733;
      AN    M      3.3;
      =     M   7004.1;
      A     L      0.1;
      BLD   102;
      L     S5T#0MS;
      SD    T    733;
      A     L      0.0;
      A(    ;
      O     DB327.DBX 1093.3;
      O     ;
      A     M   7004.2;
      AN    I      0.1;
      AN    I    180.1;
      )     ;
      =     L      0.1;
      A     L      0.1;
      A     T    734;
      AN    M      3.3;
      =     M   7004.2;
      A     L      0.1;
      BLD   102;
      L     S5T#0MS;
      SD    T    734;
      A     L      0.0;
      A(    ;
      O     DB327.DBX 1095.3;
      O     ;
      A     M   7004.3;
      AN    I      0.1;
      AN    I    180.1;
      )     ;
      =     L      0.1;
      A     L      0.1;
      A     T    735;
      AN    M      3.3;
      =     M   7004.3;
      A     L      0.1;
      BLD   102;
      L     S5T#0MS;
      SD    T    735;
      A     L      0.0;
      A(    ;
      O     DB327.DBX 1097.3;
      O     ;
      A     M   7004.4;
      AN    I      0.1;
      AN    I    180.1;
      )     ;
      =     L      0.1;
      A     L      0.1;
      A     T    736;
      AN    M      3.3;
      =     M   7004.4;
      A     L      0.1;
      BLD   102;
      L     S5T#0MS;
      SD    T    736;
      A     L      0.0;
      A(    ;
      O     DB327.DBX 1099.3;
      O     ;
      A     M   7004.5;
      AN    I      0.1;
      AN    I    180.1;
      )     ;
      =     L      0.1;
      A     L      0.1;
      A     T    737;
      AN    M      3.3;
      =     M   7004.5;
      A     L      0.1;
      BLD   102;
      L     S5T#0MS;
      SD    T    737;
      A     L      0.0;
      A(    ;
      O     DB327.DBX 1101.3;
      O     ;
      A     M   7004.6;
      AN    I      0.1;
      AN    I    180.1;
      )     ;
      =     L      0.1;
      A     L      0.1;
      A     T    738;
      AN    M      3.3;
      =     M   7004.6;
      A     L      0.1;
      BLD   102;
      L     S5T#0MS;
      SD    T    738;
      A     L      0.0;
      A(    ;
      O     DB327.DBX 1103.3;
      O     ;
      A     M   7004.7;
      AN    I      0.1;
      AN    I    180.1;
      )     ;
      =     L      0.1;
      A     L      0.1;
      A     T    739;
      AN    M      3.3;
      =     M   7004.7;
      A     L      0.1;
      BLD   102;
      L     S5T#0MS;
      SD    T    739;
NETWORK
TITLE =PROFINET ERROR(150~159)

      A     M      3.3;
      =     L      0.0;
      A     L      0.0;
      A(    ;
      O     DB327.DBX 1323.3;
      O     ;
      A     M   7018.5;
      AN    I      0.1;
      AN    I    180.1;
      )     ;
      =     L      0.1;
      A     L      0.1;
      A     T    849;
      =     M   7018.5;
      A     L      0.1;
      BLD   102;
      L     S5T#0MS;
      SD    T    849;
      A     L      0.0;
      A(    ;
      O     DB327.DBX 1325.3;
      O     ;
      A     M   7018.6;
      AN    I      0.1;
      AN    I    180.1;
      )     ;
      =     L      0.1;
      A     L      0.1;
      A     T    850;
      AN    M      3.3;
      =     M   7018.6;
      A     L      0.1;
      BLD   102;
      L     S5T#0MS;
      SD    T    850;
      A     L      0.0;
      A(    ;
      O     DB327.DBX 1327.3;
      O     ;
      A     M   7018.7;
      AN    I      0.1;
      AN    I    180.1;
      )     ;
      =     L      0.1;
      A     L      0.1;
      A     T    851;
      AN    M      3.3;
      =     M   7018.7;
      A     L      0.1;
      BLD   102;
      L     S5T#0MS;
      SD    T    851;
      A     L      0.0;
      A(    ;
      O     DB327.DBX 1329.3;
      O     ;
      A     M   7019.0;
      AN    I      0.1;
      AN    I    180.1;
      )     ;
      =     L      0.1;
      A     L      0.1;
      A     T    852;
      AN    M      3.3;
      =     M   7019.0;
      A     L      0.1;
      BLD   102;
      L     S5T#0MS;
      SD    T    852;
      A     L      0.0;
      A(    ;
      O     DB327.DBX 1331.3;
      O     ;
      A     M   7019.1;
      AN    I      0.1;
      AN    I    180.1;
      )     ;
      =     L      0.1;
      A     L      0.1;
      A     T    853;
      AN    M      3.3;
      =     M   7019.1;
      A     L      0.1;
      BLD   102;
      L     S5T#0MS;
      SD    T    853;
      A     L      0.0;
      A(    ;
      O     DB327.DBX 1333.3;
      O     ;
      A     M   7019.2;
      AN    I      0.1;
      AN    I    180.1;
      )     ;
      =     L      0.1;
      A     L      0.1;
      A     T    854;
      AN    M      3.3;
      =     M   7019.2;
      A     L      0.1;
      BLD   102;
      L     S5T#0MS;
      SD    T    854;
      A     L      0.0;
      A(    ;
      O     DB327.DBX 1335.3;
      O     ;
      A     M   7019.3;
      AN    I      0.1;
      AN    I    180.1;
      )     ;
      =     L      0.1;
      A     L      0.1;
      A     T    855;
      AN    M      3.3;
      =     M   7019.3;
      A     L      0.1;
      BLD   102;
      L     S5T#0MS;
      SD    T    855;
      A     L      0.0;
      A(    ;
      O     DB327.DBX 1337.3;
      O     ;
      A     M   7019.4;
      AN    I      0.1;
      AN    I    180.1;
      )     ;
      =     L      0.1;
      A     L      0.1;
      A     T    856;
      AN    M      3.3;
      =     M   7019.4;
      A     L      0.1;
      BLD   102;
      L     S5T#0MS;
      SD    T    856;
      A     L      0.0;
      A(    ;
      O     DB327.DBX 1339.3;
      O     ;
      A     M   7019.5;
      AN    I      0.1;
      AN    I    180.1;
      )     ;
      =     L      0.1;
      A     L      0.1;
      A     T    857;
      AN    M      3.3;
      =     M   7019.5;
      A     L      0.1;
      BLD   102;
      L     S5T#0MS;
      SD    T    857;
      A     L      0.0;
      A(    ;
      O     DB327.DBX 1341.3;
      O     ;
      A     M   7019.6;
      AN    I      0.1;
      AN    I    180.1;
      )     ;
      =     L      0.1;
      A     L      0.1;
      A     T    858;
      AN    M      3.3;
      =     M   7019.6;
      A     L      0.1;
      BLD   102;
      L     S5T#0MS;
      SD    T    858;
NETWORK
TITLE =CP TRIP(20~27)
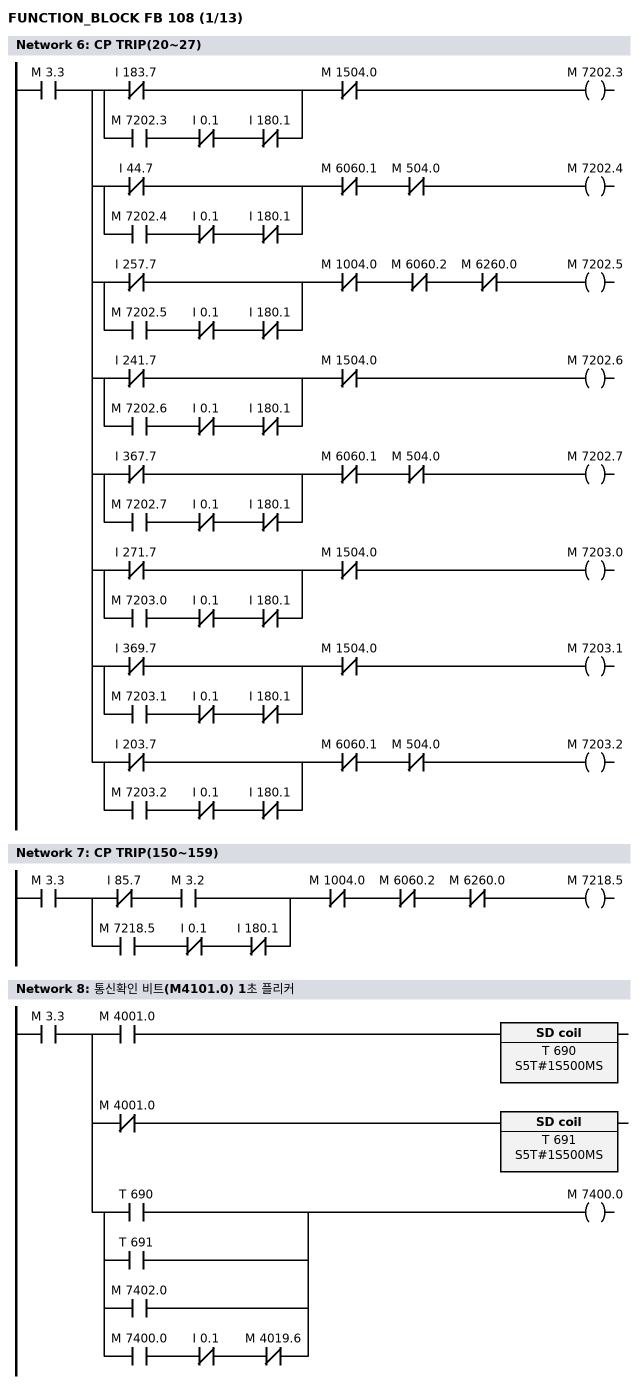

      A     M      3.3;
      =     L      0.0;
      A     L      0.0;
      A(    ;
      ON    I    183.7;
      O     ;
      A     M   7202.3;
      AN    I      0.1;
      AN    I    180.1;
      )     ;
      AN    M   1504.0;
      =     M   7202.3;
      A     L      0.0;
      A(    ;
      ON    I     44.7;
      O     ;
      A     M   7202.4;
      AN    I      0.1;
      AN    I    180.1;
      )     ;
      AN    M   6060.1;
      AN    M    504.0;
      =     M   7202.4;
      A     L      0.0;
      A(    ;
      ON    I    257.7;
      O     ;
      A     M   7202.5;
      AN    I      0.1;
      AN    I    180.1;
      )     ;
      AN    M   1004.0;
      AN    M   6060.2;
      AN    M   6260.0;
      =     M   7202.5;
      A     L      0.0;
      A(    ;
      ON    I    241.7;
      O     ;
      A     M   7202.6;
      AN    I      0.1;
      AN    I    180.1;
      )     ;
      AN    M   1504.0;
      =     M   7202.6;
      A     L      0.0;
      A(    ;
      ON    I    367.7;
      O     ;
      A     M   7202.7;
      AN    I      0.1;
      AN    I    180.1;
      )     ;
      AN    M   6060.1;
      AN    M    504.0;
      =     M   7202.7;
      A     L      0.0;
      A(    ;
      ON    I    271.7;
      O     ;
      A     M   7203.0;
      AN    I      0.1;
      AN    I    180.1;
      )     ;
      AN    M   1504.0;
      =     M   7203.0;
      A     L      0.0;
      A(    ;
      ON    I    369.7;
      O     ;
      A     M   7203.1;
      AN    I      0.1;
      AN    I    180.1;
      )     ;
      AN    M   1504.0;
      =     M   7203.1;
      A     L      0.0;
      A(    ;
      ON    I    203.7;
      O     ;
      A     M   7203.2;
      AN    I      0.1;
      AN    I    180.1;
      )     ;
      AN    M   6060.1;
      AN    M    504.0;
      =     M   7203.2;
NETWORK
TITLE =CP TRIP(150~159)

      A     M      3.3;
      A(    ;
      AN    I     85.7;
      A     M      3.2;
      O     ;
      A     M   7218.5;
      AN    I      0.1;
      AN    I    180.1;
      )     ;
      AN    M   1004.0;
      AN    M   6060.2;
      AN    M   6260.0;
      =     M   7218.5;
NETWORK
TITLE =통신확인 비트(M4101.0) 1초 플리커

      A     M      3.3;
      =     L      0.0;
      A     L      0.0;
      A     M   4001.0;
      L     S5T#1S500MS;
      SD    T    690;
      A     L      0.0;
      AN    M   4001.0;
      L     S5T#1S500MS;
      SD    T    691;
      A     L      0.0;
      A(    ;
      O     T    690;
      O     T    691;
      O     M   7402.0;
      O     ;
      A     M   7400.0;
      AN    I      0.1;
      AN    M   4019.6;
      )     ;
      =     M   7400.0;
NETWORK
TITLE =제어반 허브1 알람
